LIN {X 0,Y 611.244,Z 977.53,A -85,B 0,C 180,E1 7676.81,E2 7676.81} C_VEL
LIN {X 0,Y 611.181,Z 977.53,A -85,B 0,C 180,E1 7682.54,E2 7682.54} C_VEL
LIN {X 0,Y 611.095,Z 977.53,A -85,B 0,C 180,E1 7688.3,E2 7688.3} C_VEL
LIN {X 0,Y 611.106,Z 977.53,A -85,B 0,C 180,E1 7694.015,E2 7694.015} C_VEL
LIN {X 0,Y 611.087,Z 977.53,A -85,B 0,C 180,E1 7700.225,E2 7700.225} C_VEL
LIN {X 0,Y 611.05,Z 977.53,A -85,B 0,C 180,E1 7705.218,E2 7705.218} C_VEL
LIN {X 0,Y 611.356,Z 977.53,A -85,B 0,C 180,E1 7711.287,E2 7711.287} C_VEL
LIN {X 0,Y 625.159,Z 1016.829,A -85,B 0,C 180,E1 7712.531,E2 7712.531} C_VEL
LIN {X 0,Y 623.748,Z 1056.325,A -85,B 0,C 180,E1 7713.584,E2 7713.584} C_VEL
LIN {X 0,Y 621.786,Z 1092.605,A -85,B 0,C 180,E1 7715.073,E2 7715.073} C_VEL
LIN {X 0,Y 619.511,Z 1127.087,A -85,B 0,C 180,E1 7717.049,E2 7717.049} C_VEL
LIN {X 0,Y 617.19,Z 1158.439,A -85,B 0,C 180,E1 7719.455,E2 7719.455} C_VEL
LIN {X 0,Y 615.112,Z 1187.568,A -85,B 0,C 180,E1 7722.428,E2 7722.428} C_VEL
LIN {X 0,Y 613.624,Z 1211.374,A -85,B 0,C 180,E1 7725.695,E2 7725.695} C_VEL
LIN {X 0,Y 612.633,Z 1230.256,A -85,B 0,C 180,E1 7729.301,E2 7729.301} C_VEL
LIN {X 0,Y 612.205,Z 1242.892,A -85,B 0,C 180,E1 7732.882,E2 7732.882} C_VEL
LIN {X 0,Y 612.031,Z 1249.086,A -85,B 0,C 180,E1 7735.731,E2 7735.731} C_VEL
LIN {X 0,Y 612.003,Z 1252.15,A -85,B 0,C 180,E1 7738.571,E2 7738.571} C_VEL
LIN {X 0,Y 612.141,Z 1252.095,A -85,B 0,C 180,E1 7741.408,E2 7741.408} C_VEL
LIN {X 0,Y 612.201,Z 1247.774,A -85,B 0,C 180,E1 7744.959,E2 7744.959} C_VEL
LIN {X 0,Y 612.397,Z 1238.388,A -85,B 0,C 180,E1 7748.526,E2 7748.526} C_VEL
LIN {X 0,Y 612.998,Z 1222.369,A -85,B 0,C 180,E1 7752.291,E2 7752.291} C_VEL
LIN {X 0,Y 614.182,Z 1202.539,A -85,B 0,C 180,E1 7755.551,E2 7755.551} C_VEL
LIN {X 0,Y 615.818,Z 1177.097,A -85,B 0,C 180,E1 7758.642,E2 7758.642} C_VEL
LIN {X 0,Y 617.854,Z 1148.189,A -85,B 0,C 180,E1 7761.28,E2 7761.28} C_VEL
LIN {X 0,Y 620.03,Z 1114.997,A -85,B 0,C 180,E1 7763.553,E2 7763.553} C_VEL
LIN {X 0,Y 622.154,Z 1077.81,A -85,B 0,C 180,E1 7765.402,E2 7765.402} C_VEL
LIN {X 0,Y 623.879,Z 1037.397,A -85,B 0,C 180,E1 7766.756,E2 7766.756} C_VEL
LIN {X 0,Y 623.911,Z 1015.287,A -85,B 0,C 180,E1 7767.268,E2 7767.268} C_VEL
LIN {X 0,Y 611.262,Z 977.53,A -85,B 0,C 180,E1 7768.438,E2 7768.438} C_VEL
LIN {X 0,Y 611.055,Z 977.53,A -85,B 0,C 180,E1 7774.047,E2 7774.047} C_VEL
LIN {X 0,Y 607.146,Z 977.53,A -85,B 0,C 180,E1 7775.649,E2 7775.649} C_VEL
LIN {X 0,Y 603.114,Z 977.53,A -85,B 0,C 180,E1 7777.271,E2 7777.271} C_VEL
LIN {X 0,Y 602.965,Z 977.53,A -85,B 0,C 180,E1 7783.226,E2 7783.226} C_VEL
LIN {X 0,Y 603.021,Z 977.53,A -85,B 0,C 180,E1 7789.216,E2 7789.216} C_VEL
LIN {X 0,Y 603.25,Z 977.53,A -85,B 0,C 180,E1 7794.718,E2 7794.718} C_VEL
LIN {X 0,Y 603.286,Z 978.056,A -85,B 0,C 180,E1 7798.731,E2 7798.731} C_VEL
LIN {X 0,Y 614.334,Z 1020.655,A -85,B 0,C 180,E1 7801.57,E2 7801.57} C_VEL
LIN {X 0,Y 617.712,Z 1027.362,A -85,B 0,C 180,E1 7801.794,E2 7801.794} C_VEL
LIN {X 0,Y 616.69,Z 1077.628,A -85,B 0,C 180,E1 7802.575,E2 7802.575} C_VEL
LIN {X 0,Y 614.875,Z 1118.446,A -85,B 0,C 180,E1 7803.772,E2 7803.772} C_VEL
LIN {X 0,Y 612.716,Z 1155.496,A -85,B 0,C 180,E1 7805.411,E2 7805.411} C_VEL
LIN {X 0,Y 610.412,Z 1190.848,A -85,B 0,C 180,E1 7807.57,E2 7807.57} C_VEL
LIN {X 0,Y 608.203,Z 1224.713,A -85,B 0,C 180,E1 7810.353,E2 7810.353} C_VEL
LIN {X 0,Y 606.411,Z 1253.135,A -85,B 0,C 180,E1 7813.494,E2 7813.494} C_VEL
LIN {X 0,Y 605.216,Z 1275.601,A -85,B 0,C 180,E1 7816.8,E2 7816.8} C_VEL
LIN {X 0,Y 604.571,Z 1292.527,A -85,B 0,C 180,E1 7820.267,E2 7820.267} C_VEL
LIN {X 0,Y 604.307,Z 1303.392,A -85,B 0,C 180,E1 7823.528,E2 7823.528} C_VEL
LIN {X 0,Y 604.191,Z 1310.148,A -85,B 0,C 180,E1 7827.132,E2 7827.132} C_VEL
LIN {X 0,Y 604.162,Z 1311.816,A -85,B 0,C 180,E1 7830.007,E2 7830.007} C_VEL
LIN {X 0,Y 604.16,Z 1309.117,A -85,B 0,C 180,E1 7833.602,E2 7833.602} C_VEL
LIN {X 0,Y 604.353,Z 1301.231,A -85,B 0,C 180,E1 7837.208,E2 7837.208} C_VEL
LIN {X 0,Y 604.717,Z 1289.245,A -85,B 0,C 180,E1 7840.474,E2 7840.474} C_VEL
LIN {X 0,Y 605.539,Z 1270.525,A -85,B 0,C 180,E1 7843.944,E2 7843.944} C_VEL
LIN {X 0,Y 606.897,Z 1245.039,A -85,B 0,C 180,E1 7847.441,E2 7847.441} C_VEL
LIN {X 0,Y 608.897,Z 1215.102,A -85,B 0,C 180,E1 7850.51,E2 7850.51} C_VEL
LIN {X 0,Y 611.057,Z 1182.798,A -85,B 0,C 180,E1 7852.996,E2 7852.996} C_VEL
LIN {X 0,Y 613.398,Z 1147.018,A -85,B 0,C 180,E1 7855.041,E2 7855.041} C_VEL
LIN {X 0,Y 615.534,Z 1108.168,A -85,B 0,C 180,E1 7856.605,E2 7856.605} C_VEL
LIN {X 0,Y 617.049,Z 1069.386,A -85,B 0,C 180,E1 7857.595,E2 7857.595} C_VEL
LIN {X 0,Y 617.131,Z 1025.386,A -85,B 0,C 180,E1 7858.25,E2 7858.25} C_VEL
LIN {X 0,Y 609.111,Z 1006.368,A -85,B 0,C 180,E1 7858.929,E2 7858.929} C_VEL
LIN {X 0,Y 603.325,Z 977.53,A -85,B 0,C 180,E1 7860.768,E2 7860.768} C_VEL
LIN {X 0,Y 603.185,Z 977.53,A -85,B 0,C 180,E1 7866.525,E2 7866.525} C_VEL
LIN {X 0,Y 603.127,Z 977.53,A -85,B 0,C 180,E1 7871.111,E2 7871.111} C_VEL
LIN {X 0,Y 603.121,Z 977.53,A -85,B 0,C 180,E1 7876.778,E2 7876.778} C_VEL
LIN {X 0,Y 603.127,Z 977.53,A -85,B 0,C 180,E1 7881.164,E2 7881.164} C_VEL
LIN {X 0,Y 603.141,Z 977.53,A -85,B 0,C 180,E1 7886.464,E2 7886.464} C_VEL
LIN {X 0,Y 603.328,Z 977.53,A -85,B 0,C 180,E1 7891.539,E2 7891.539} C_VEL
LIN {X 0,Y 603.432,Z 977.53,A -85,B 0,C 180,E1 7896.325,E2 7896.325} C_VEL
LIN {X 0,Y 603.526,Z 977.53,A -85,B 0,C 180,E1 7900.963,E2 7900.963} C_VEL
LIN {X 0,Y 603.545,Z 977.53,A -85,B 0,C 180,E1 7905.472,E2 7905.472} C_VEL
LIN {X 0,Y 603.751,Z 977.53,A -85,B 0,C 180,E1 7911.351,E2 7911.351} C_VEL
LIN {X 0,Y 603.871,Z 977.53,A -85,B 0,C 180,E1 7913.437,E2 7913.437} C_VEL
LIN {X 0,Y 611.206,Z 1003.096,A -85,B 0,C 180,E1 7914.239,E2 7914.239} C_VEL
LIN {X 0,Y 610.052,Z 1060.493,A -85,B 0,C 180,E1 7915.336,E2 7915.336} C_VEL
LIN {X 0,Y 609.176,Z 1088.907,A -85,B 0,C 180,E1 7916.445,E2 7916.445} C_VEL
LIN {X 0,Y 608.114,Z 1114.127,A -85,B 0,C 180,E1 7918.047,E2 7918.047} C_VEL
LIN {X 0,Y 606.979,Z 1135.109,A -85,B 0,C 180,E1 7920.01,E2 7920.01} C_VEL
LIN {X 0,Y 606.057,Z 1152.124,A -85,B 0,C 180,E1 7922.338,E2 7922.338} C_VEL
LIN {X 0,Y 605.342,Z 1164.6,A -85,B 0,C 180,E1 7925.036,E2 7925.036} C_VEL
LIN {X 0,Y 605.013,Z 1170.296,A -85,B 0,C 180,E1 7927.203,E2 7927.203} C_VEL
LIN {X 0,Y 604.838,Z 1172.559,A -85,B 0,C 180,E1 7930.109,E2 7930.109} C_VEL
LIN {X 0,Y 604.97,Z 1168.797,A -85,B 0,C 180,E1 7933.037,E2 7933.037} C_VEL
LIN {X 0,Y 605.309,Z 1159.648,A -85,B 0,C 180,E1 7935.744,E2 7935.744} C_VEL
LIN {X 0,Y 605.903,Z 1145.613,A -85,B 0,C 180,E1 7938.203,E2 7938.203} C_VEL
LIN {X 0,Y 606.787,Z 1126.099,A -85,B 0,C 180,E1 7940.472,E2 7940.472} C_VEL
LIN {X 0,Y 607.731,Z 1102.106,A -85,B 0,C 180,E1 7942.367,E2 7942.367} C_VEL
LIN {X 0,Y 608.82,Z 1074.436,A -85,B 0,C 180,E1 7943.782,E2 7943.782} C_VEL
LIN {X 0,Y 609.304,Z 1045.453,A -85,B 0,C 180,E1 7944.644,E2 7944.644} C_VEL
LIN {X 0,Y 609.265,Z 999.333,A -85,B 0,C 180,E1 7945.356,E2 7945.356} C_VEL
LIN {X 0,Y 603.556,Z 977.53,A -85,B 0,C 180,E1 7945.917,E2 7945.917} C_VEL
LIN {X 0,Y 603.26,Z 977.53,A -85,B 0,C 180,E1 7951.843,E2 7951.843} C_VEL
LIN {X 0,Y 603.173,Z 977.53,A -85,B 0,C 180,E1 7957.087,E2 7957.087} C_VEL
LIN {X 0,Y 603.145,Z 977.53,A -85,B 0,C 180,E1 7962.72,E2 7962.72} C_VEL
LIN {X 0,Y 603.092,Z 977.53,A -85,B 0,C 180,E1 7967.274,E2 7967.274} C_VEL
LIN {X 0,Y 603.118,Z 977.53,A -85,B 0,C 180,E1 7972.909,E2 7972.909} C_VEL
LIN {X 0,Y 603.263,Z 977.53,A -85,B 0,C 180,E1 7978.659,E2 7978.659} C_VEL
LIN {X 0,Y 603.392,Z 977.53,A -85,B 0,C 180,E1 7983.119,E2 7983.119} C_VEL
LIN {X 0,Y 603.49,Z 977.53,A -85,B 0,C 180,E1 7988.291,E2 7988.291} C_VEL
LIN {X 0,Y 603.561,Z 977.53,A -85,B 0,C 180,E1 7993.962,E2 7993.962} C_VEL
LIN {X 0,Y 603.681,Z 977.53,A -85,B 0,C 180,E1 7999.874,E2 7999.874} C_VEL
LIN {X 0,Y 603.86,Z 977.53,A -85,B 0,C 180,E1 8004.233,E2 8004.233} C_VEL
LIN {X 0,Y 603.917,Z 977.53,A -85,B 0,C 180,E1 8008.556,E2 8008.556} C_VEL
LIN {X 0,Y 603.938,Z 977.53,A -85,B 0,C 180,E1 8012.87,E2 8012.87} C_VEL
LIN {X 0,Y 603.718,Z 977.53,A -85,B 0,C 180,E1 8017.203,E2 8017.203} C_VEL
LIN {X 0,Y 603.623,Z 977.53,A -85,B 0,C 180,E1 8023.05,E2 8023.05} C_VEL
LIN {X 0,Y 603.572,Z 977.53,A -85,B 0,C 180,E1 8027.526,E2 8027.526} C_VEL
LIN {X 0,Y 603.428,Z 977.53,A -85,B 0,C 180,E1 8032.12,E2 8032.12} C_VEL
LIN {X 0,Y 603.363,Z 977.53,A -85,B 0,C 180,E1 8036.867,E2 8036.867} C_VEL
LIN {X 0,Y 603.267,Z 977.53,A -85,B 0,C 180,E1 8041.827,E2 8041.827} C_VEL
LIN {X 0,Y 603.174,Z 977.53,A -85,B 0,C 180,E1 8047.071,E2 8047.071} C_VEL
LIN {X 0,Y 603.135,Z 977.53,A -85,B 0,C 180,E1 8052.704,E2 8052.704} C_VEL
LIN {X 0,Y 603.086,Z 977.53,A -85,B 0,C 180,E1 8057.275,E2 8057.275} C_VEL
LIN {X 0,Y 603.127,Z 977.53,A -85,B 0,C 180,E1 8062.91,E2 8062.91} C_VEL
LIN {X 0,Y 603.264,Z 977.53,A -85,B 0,C 180,E1 8068.637,E2 8068.637} C_VEL
LIN {X 0,Y 603.415,Z 977.689,A -85,B 0,C 180,E1 8070.929,E2 8070.929} C_VEL
LIN {X 0,Y 617.942,Z 1019.384,A -85,B 0,C 180,E1 8072.271,E2 8072.271} C_VEL
LIN {X 0,Y 616.402,Z 1059.794,A -85,B 0,C 180,E1 8073.401,E2 8073.401} C_VEL
LIN {X 0,Y 614.144,Z 1097.737,A -85,B 0,C 180,E1 8075.035,E2 8075.035} C_VEL
LIN {X 0,Y 611.585,Z 1133.527,A -85,B 0,C 180,E1 8077.216,E2 8077.216} C_VEL
LIN {X 0,Y 609.219,Z 1164.975,A -85,B 0,C 180,E1 8079.804,E2 8079.804} C_VEL
LIN {X 0,Y 607.126,Z 1192.049,A -85,B 0,C 180,E1 8082.751,E2 8082.751} C_VEL
LIN {X 0,Y 605.697,Z 1213.671,A -85,B 0,C 180,E1 8085.873,E2 8085.873} C_VEL
LIN {X 0,Y 604.809,Z 1230.485,A -85,B 0,C 180,E1 8089.161,E2 8089.161} C_VEL
LIN {X 0,Y 604.345,Z 1243.19,A -85,B 0,C 180,E1 8092.789,E2 8092.789} C_VEL
LIN {X 0,Y 604.146,Z 1249.426,A -85,B 0,C 180,E1 8095.675,E2 8095.675} C_VEL
LIN {X 0,Y 604.112,Z 1252.516,A -85,B 0,C 180,E1 8098.553,E2 8098.553} C_VEL
LIN {X 0,Y 604.266,Z 1252.471,A -85,B 0,C 180,E1 8101.426,E2 8101.426} C_VEL
LIN {X 0,Y 604.313,Z 1248.139,A -85,B 0,C 180,E1 8105.024,E2 8105.024} C_VEL
LIN {X 0,Y 604.545,Z 1238.716,A -85,B 0,C 180,E1 8108.638,E2 8108.638} C_VEL
LIN {X 0,Y 605.162,Z 1223.209,A -85,B 0,C 180,E1 8112.336,E2 8112.336} C_VEL
LIN {X 0,Y 606.453,Z 1202.656,A -85,B 0,C 180,E1 8115.754,E2 8115.754} C_VEL
LIN {X 0,Y 608.146,Z 1177.906,A -85,B 0,C 180,E1 8118.792,E2 8118.792} C_VEL
LIN {X 0,Y 610.342,Z 1148.346,A -85,B 0,C 180,E1 8121.519,E2 8121.519} C_VEL
LIN {X 0,Y 612.598,Z 1114.641,A -85,B 0,C 180,E1 8123.844,E2 8123.844} C_VEL
LIN {X 0,Y 614.838,Z 1077.728,A -85,B 0,C 180,E1 8125.689,E2 8125.689} C_VEL
LIN {X 0,Y 616.627,Z 1037.109,A -85,B 0,C 180,E1 8127.056,E2 8127.056} C_VEL
LIN {X 0,Y 616.657,Z 1017.258,A -85,B 0,C 180,E1 8127.528,E2 8127.528} C_VEL
LIN {X 0,Y 603.35,Z 977.53,A -85,B 0,C 180,E1 8128.823,E2 8128.823} C_VEL
LIN {X 0,Y 603.163,Z 977.53,A -85,B 0,C 180,E1 8134.041,E2 8134.041} C_VEL
LIN {X 0,Y 603.114,Z 977.53,A -85,B 0,C 180,E1 8137.271,E2 8137.271} C_VEL
LIN {X 0,Y 599.073,Z 977.53,A -85,B 0,C 180,E1 8138.893,E2 8138.893} C_VEL
LIN {X 0,Y 595.066,Z 977.53,A -85,B 0,C 180,E1 8140.535,E2 8140.535} C_VEL
LIN {X 0,Y 595.061,Z 977.53,A -85,B 0,C 180,E1 8145.457,E2 8145.457} C_VEL
LIN {X 0,Y 595.116,Z 977.53,A -85,B 0,C 180,E1 8150.474,E2 8150.474} C_VEL
LIN {X 0,Y 595.331,Z 977.53,A -85,B 0,C 180,E1 8155.956,E2 8155.956} C_VEL
LIN {X 0,Y 595.329,Z 977.778,A -85,B 0,C 180,E1 8158.372,E2 8158.372} C_VEL
LIN {X 0,Y 606.071,Z 1020.674,A -85,B 0,C 180,E1 8161.23,E2 8161.23} C_VEL
LIN {X 0,Y 610.515,Z 1031.2,A -85,B 0,C 180,E1 8161.553,E2 8161.553} C_VEL
LIN {X 0,Y 609.35,Z 1077.574,A -85,B 0,C 180,E1 8162.301,E2 8162.301} C_VEL
LIN {X 0,Y 607.51,Z 1117.465,A -85,B 0,C 180,E1 8163.485,E2 8163.485} C_VEL
LIN {X 0,Y 605.122,Z 1155.894,A -85,B 0,C 180,E1 8165.209,E2 8165.209} C_VEL
LIN {X 0,Y 602.651,Z 1191.864,A -85,B 0,C 180,E1 8167.461,E2 8167.461} C_VEL
LIN {X 0,Y 600.576,Z 1223.393,A -85,B 0,C 180,E1 8170.093,E2 8170.093} C_VEL
LIN {X 0,Y 598.666,Z 1251.991,A -85,B 0,C 180,E1 8173.274,E2 8173.274} C_VEL
LIN {X 0,Y 597.407,Z 1274.588,A -85,B 0,C 180,E1 8176.625,E2 8176.625} C_VEL
LIN {X 0,Y 596.722,Z 1291.588,A -85,B 0,C 180,E1 8180.137,E2 8180.137} C_VEL
LIN {X 0,Y 596.439,Z 1302.503,A -85,B 0,C 180,E1 8183.442,E2 8183.442} C_VEL
LIN {X 0,Y 596.341,Z 1309.289,A -85,B 0,C 180,E1 8187.094,E2 8187.094} C_VEL
LIN {X 0,Y 596.316,Z 1310.95,A -85,B 0,C 180,E1 8190.007,E2 8190.007} C_VEL
LIN {X 0,Y 596.322,Z 1308.212,A -85,B 0,C 180,E1 8193.649,E2 8193.649} C_VEL
LIN {X 0,Y 596.524,Z 1300.246,A -85,B 0,C 180,E1 8197.304,E2 8197.304} C_VEL
LIN {X 0,Y 596.853,Z 1288.156,A -85,B 0,C 180,E1 8200.613,E2 8200.613} C_VEL
LIN {X 0,Y 597.753,Z 1267.354,A -85,B 0,C 180,E1 8204.504,E2 8204.504} C_VEL
LIN {X 0,Y 599.211,Z 1243.275,A -85,B 0,C 180,E1 8207.81,E2 8207.81} C_VEL
LIN {X 0,Y 601.274,Z 1213.743,A -85,B 0,C 180,E1 8210.833,E2 8210.833} C_VEL
LIN {X 0,Y 603.708,Z 1180.457,A -85,B 0,C 180,E1 8213.391,E2 8213.391} C_VEL
LIN {X 0,Y 606.121,Z 1145.205,A -85,B 0,C 180,E1 8215.399,E2 8215.399} C_VEL
LIN {X 0,Y 608.335,Z 1106.849,A -85,B 0,C 180,E1 8216.939,E2 8216.939} C_VEL
LIN {X 0,Y 609.968,Z 1067.091,A -85,B 0,C 180,E1 8217.943,E2 8217.943} C_VEL
LIN {X 0,Y 610.095,Z 1027.985,A -85,B 0,C 180,E1 8218.527,E2 8218.527} C_VEL
LIN {X 0,Y 600.85,Z 1004.137,A -85,B 0,C 180,E1 8219.353,E2 8219.353} C_VEL
LIN {X 0,Y 595.426,Z 977.53,A -85,B 0,C 180,E1 8221.124,E2 8221.124} C_VEL
LIN {X 0,Y 595.257,Z 977.53,A -85,B 0,C 180,E1 8225.845,E2 8225.845} C_VEL
LIN {X 0,Y 595.206,Z 977.53,A -85,B 0,C 180,E1 8231.454,E2 8231.454} C_VEL
LIN {X 0,Y 595.22,Z 977.53,A -85,B 0,C 180,E1 8236.6,E2 8236.6} C_VEL
LIN {X 0,Y 595.155,Z 977.53,A -85,B 0,C 180,E1 8242.354,E2 8242.354} C_VEL
LIN {X 0,Y 595.256,Z 977.53,A -85,B 0,C 180,E1 8247.702,E2 8247.702} C_VEL
LIN {X 0,Y 595.492,Z 977.53,A -85,B 0,C 180,E1 8252.963,E2 8252.963} C_VEL
LIN {X 0,Y 595.526,Z 977.53,A -85,B 0,C 180,E1 8257.577,E2 8257.577} C_VEL
LIN {X 0,Y 595.598,Z 977.53,A -85,B 0,C 180,E1 8262.237,E2 8262.237} C_VEL
LIN {X 0,Y 595.618,Z 977.53,A -85,B 0,C 180,E1 8266.776,E2 8266.776} C_VEL
LIN {X 0,Y 595.916,Z 977.53,A -85,B 0,C 180,E1 8272.707,E2 8272.707} C_VEL
LIN {X 0,Y 595.959,Z 977.53,A -85,B 0,C 180,E1 8273.075,E2 8273.075} C_VEL
LIN {X 0,Y 603.888,Z 1005.096,A -85,B 0,C 180,E1 8273.984,E2 8273.984} C_VEL
LIN {X 0,Y 602.566,Z 1062.313,A -85,B 0,C 180,E1 8275.126,E2 8275.126} C_VEL
LIN {X 0,Y 601.696,Z 1089.668,A -85,B 0,C 180,E1 8276.22,E2 8276.22} C_VEL
LIN {X 0,Y 600.541,Z 1114.948,A -85,B 0,C 180,E1 8277.842,E2 8277.842} C_VEL
LIN {X 0,Y 599.239,Z 1137.543,A -85,B 0,C 180,E1 8280.01,E2 8280.01} C_VEL
LIN {X 0,Y 598.228,Z 1154.978,A -85,B 0,C 180,E1 8282.551,E2 8282.551} C_VEL
LIN {X 0,Y 597.515,Z 1166.087,A -85,B 0,C 180,E1 8285.102,E2 8285.102} C_VEL
LIN {X 0,Y 597.169,Z 1171.546,A -85,B 0,C 180,E1 8287.298,E2 8287.298} C_VEL
LIN {X 0,Y 596.991,Z 1173.453,A -85,B 0,C 180,E1 8290.244,E2 8290.244} C_VEL
LIN {X 0,Y 597.158,Z 1169.391,A -85,B 0,C 180,E1 8293.21,E2 8293.21} C_VEL
LIN {X 0,Y 597.519,Z 1159.721,A -85,B 0,C 180,E1 8295.984,E2 8295.984} C_VEL
LIN {X 0,Y 598.219,Z 1144.574,A -85,B 0,C 180,E1 8298.565,E2 8298.565} C_VEL
LIN {X 0,Y 599.174,Z 1124.452,A -85,B 0,C 180,E1 8300.841,E2 8300.841} C_VEL
LIN {X 0,Y 600.182,Z 1100.359,A -85,B 0,C 180,E1 8302.682,E2 8302.682} C_VEL
LIN {X 0,Y 601.226,Z 1072.101,A -85,B 0,C 180,E1 8304.086,E2 8304.086} C_VEL
LIN {X 0,Y 601.73,Z 1041.841,A -85,B 0,C 180,E1 8304.921,E2 8304.921} C_VEL
LIN {X 0,Y 601.803,Z 1001.087,A -85,B 0,C 180,E1 8305.551,E2 8305.551} C_VEL
LIN {X 0,Y 595.614,Z 977.53,A -85,B 0,C 180,E1 8306.157,E2 8306.157} C_VEL
LIN {X 0,Y 595.293,Z 977.53,A -85,B 0,C 180,E1 8312.32,E2 8312.32} C_VEL
LIN {X 0,Y 595.207,Z 977.53,A -85,B 0,C 180,E1 8317.879,E2 8317.879} C_VEL
LIN {X 0,Y 595.266,Z 977.53,A -85,B 0,C 180,E1 8323.424,E2 8323.424} C_VEL
LIN {X 0,Y 595.15,Z 977.53,A -85,B 0,C 180,E1 8328.541,E2 8328.541} C_VEL
LIN {X 0,Y 595.211,Z 977.53,A -85,B 0,C 180,E1 8334.56,E2 8334.56} C_VEL
LIN {X 0,Y 595.367,Z 977.53,A -85,B 0,C 180,E1 8339.93,E2 8339.93} C_VEL
LIN {X 0,Y 595.493,Z 977.53,A -85,B 0,C 180,E1 8344.362,E2 8344.362} C_VEL
LIN {X 0,Y 595.552,Z 977.53,A -85,B 0,C 180,E1 8349.126,E2 8349.126} C_VEL
LIN {X 0,Y 595.639,Z 977.53,A -85,B 0,C 180,E1 8353.743,E2 8353.743} C_VEL
LIN {X 0,Y 595.789,Z 977.53,A -85,B 0,C 180,E1 8359.738,E2 8359.738} C_VEL
LIN {X 0,Y 595.949,Z 977.53,A -85,B 0,C 180,E1 8364.156,E2 8364.156} C_VEL
LIN {X 0,Y 596.016,Z 977.53,A -85,B 0,C 180,E1 8368.536,E2 8368.536} C_VEL
LIN {X 0,Y 596.034,Z 977.53,A -85,B 0,C 180,E1 8372.908,E2 8372.908} C_VEL
LIN {X 0,Y 595.818,Z 977.53,A -85,B 0,C 180,E1 8377.299,E2 8377.299} C_VEL
LIN {X 0,Y 595.752,Z 977.53,A -85,B 0,C 180,E1 8381.733,E2 8381.733} C_VEL
LIN {X 0,Y 595.657,Z 977.53,A -85,B 0,C 180,E1 8386.243,E2 8386.243} C_VEL
LIN {X 0,Y 595.544,Z 977.53,A -85,B 0,C 180,E1 8390.86,E2 8390.86} C_VEL
LIN {X 0,Y 595.44,Z 977.53,A -85,B 0,C 180,E1 8395.626,E2 8395.626} C_VEL
LIN {X 0,Y 595.346,Z 977.53,A -85,B 0,C 180,E1 8400.592,E2 8400.592} C_VEL
LIN {X 0,Y 595.271,Z 977.53,A -85,B 0,C 180,E1 8405.827,E2 8405.827} C_VEL
LIN {X 0,Y 595.217,Z 977.53,A -85,B 0,C 180,E1 8411.435,E2 8411.435} C_VEL
LIN {X 0,Y 595.205,Z 977.53,A -85,B 0,C 180,E1 8416.57,E2 8416.57} C_VEL
LIN {X 0,Y 595.161,Z 977.53,A -85,B 0,C 180,E1 8422.328,E2 8422.328} C_VEL
LIN {X 0,Y 595.258,Z 977.53,A -85,B 0,C 180,E1 8427.677,E2 8427.677} C_VEL
LIN {X 0,Y 595.484,Z 978.235,A -85,B 0,C 180,E1 8430.561,E2 8430.561} C_VEL
LIN {X 0,Y 610.794,Z 1020.179,A -85,B 0,C 180,E1 8431.972,E2 8431.972} C_VEL
LIN {X 0,Y 609.136,Z 1060.705,A -85,B 0,C 180,E1 8433.125,E2 8433.125} C_VEL
LIN {X 0,Y 606.683,Z 1100.08,A -85,B 0,C 180,E1 8434.867,E2 8434.867} C_VEL
LIN {X 0,Y 603.985,Z 1135.793,A -85,B 0,C 180,E1 8437.108,E2 8437.108} C_VEL
LIN {X 0,Y 601.486,Z 1166.793,A -85,B 0,C 180,E1 8439.725,E2 8439.725} C_VEL
LIN {X 0,Y 599.341,Z 1193.534,A -85,B 0,C 180,E1 8442.71,E2 8442.71} C_VEL
LIN {X 0,Y 597.772,Z 1215.966,A -85,B 0,C 180,E1 8446.057,E2 8446.057} C_VEL
LIN {X 0,Y 596.898,Z 1232.234,A -85,B 0,C 180,E1 8449.385,E2 8449.385} C_VEL
LIN {X 0,Y 596.484,Z 1243.49,A -85,B 0,C 180,E1 8452.693,E2 8452.693} C_VEL
LIN {X 0,Y 596.26,Z 1249.76,A -85,B 0,C 180,E1 8455.618,E2 8455.618} C_VEL
LIN {X 0,Y 596.22,Z 1252.88,A -85,B 0,C 180,E1 8458.533,E2 8458.533} C_VEL
LIN {X 0,Y 596.374,Z 1252.848,A -85,B 0,C 180,E1 8461.445,E2 8461.445} C_VEL
LIN {X 0,Y 596.441,Z 1248.502,A -85,B 0,C 180,E1 8465.09,E2 8465.09} C_VEL
LIN {X 0,Y 596.68,Z 1239.038,A -85,B 0,C 180,E1 8468.753,E2 8468.753} C_VEL
LIN {X 0,Y 597.347,Z 1223.864,A -85,B 0,C 180,E1 8472.419,E2 8472.419} C_VEL
LIN {X 0,Y 598.7,Z 1203.041,A -85,B 0,C 180,E1 8475.923,E2 8475.923} C_VEL
LIN {X 0,Y 600.471,Z 1178.109,A -85,B 0,C 180,E1 8479.014,E2 8479.014} C_VEL
LIN {X 0,Y 602.798,Z 1148.747,A -85,B 0,C 180,E1 8481.747,E2 8481.747} C_VEL
LIN {X 0,Y 605.16,Z 1115.407,A -85,B 0,C 180,E1 8484.077,E2 8484.077} C_VEL
LIN {X 0,Y 607.558,Z 1077.623,A -85,B 0,C 180,E1 8485.989,E2 8485.989} C_VEL
LIN {X 0,Y 609.443,Z 1036.846,A -85,B 0,C 180,E1 8487.368,E2 8487.368} C_VEL
LIN {X 0,Y 609.292,Z 1018.723,A -85,B 0,C 180,E1 8487.817,E2 8487.817} C_VEL
LIN {X 0,Y 595.404,Z 977.53,A -85,B 0,C 180,E1 8489.232,E2 8489.232} C_VEL
LIN {X 0,Y 595.264,Z 977.53,A -85,B 0,C 180,E1 8494.04,E2 8494.04} C_VEL
LIN {X 0,Y 595.122,Z 977.53,A -85,B 0,C 180,E1 8499.515,E2 8499.515} C_VEL
LIN {X 0,Y 595.066,Z 977.53,A -85,B 0,C 180,E1 8500.535,E2 8500.535} C_VEL
LIN {X 0,Y 591.085,Z 977.53,A -85,B 0,C 180,E1 8502.178,E2 8502.178} C_VEL
LIN {X 0,Y 587.14,Z 977.53,A -85,B 0,C 180,E1 8503.843,E2 8503.843} C_VEL
LIN {X 0,Y 587.203,Z 977.53,A -85,B 0,C 180,E1 8509.835,E2 8509.835} C_VEL
LIN {X 0,Y 587.423,Z 977.53,A -85,B 0,C 180,E1 8515.605,E2 8515.605} C_VEL
LIN {X 0,Y 587.468,Z 978.239,A -85,B 0,C 180,E1 8518.056,E2 8518.056} C_VEL
LIN {X 0,Y 597.814,Z 1020.503,A -85,B 0,C 180,E1 8520.88,E2 8520.88} C_VEL
LIN {X 0,Y 603.229,Z 1033.307,A -85,B 0,C 180,E1 8521.284,E2 8521.284} C_VEL
LIN {X 0,Y 601.982,Z 1078.358,A -85,B 0,C 180,E1 8522.04,E2 8522.04} C_VEL
LIN {X 0,Y 600.052,Z 1117.57,A -85,B 0,C 180,E1 8523.234,E2 8523.234} C_VEL
LIN {X 0,Y 597.545,Z 1155.69,A -85,B 0,C 180,E1 8524.973,E2 8524.973} C_VEL
LIN {X 0,Y 595.104,Z 1190.725,A -85,B 0,C 180,E1 8527.189,E2 8527.189} C_VEL
LIN {X 0,Y 592.88,Z 1222.045,A -85,B 0,C 180,E1 8529.824,E2 8529.824} C_VEL
LIN {X 0,Y 591.005,Z 1249.369,A -85,B 0,C 180,E1 8532.859,E2 8532.859} C_VEL
LIN {X 0,Y 589.653,Z 1272.508,A -85,B 0,C 180,E1 8536.256,E2 8536.256} C_VEL
LIN {X 0,Y 588.917,Z 1289.152,A -85,B 0,C 180,E1 8539.631,E2 8539.631} C_VEL
LIN {X 0,Y 588.582,Z 1301.614,A -85,B 0,C 180,E1 8543.354,E2 8543.354} C_VEL
LIN {X 0,Y 588.49,Z 1308.43,A -85,B 0,C 180,E1 8547.055,E2 8547.055} C_VEL
LIN {X 0,Y 588.491,Z 1310.085,A -85,B 0,C 180,E1 8550.007,E2 8550.007} C_VEL
LIN {X 0,Y 588.488,Z 1307.312,A -85,B 0,C 180,E1 8553.698,E2 8553.698} C_VEL
LIN {X 0,Y 588.682,Z 1299.282,A -85,B 0,C 180,E1 8557.401,E2 8557.401} C_VEL
LIN {X 0,Y 589.042,Z 1285.709,A -85,B 0,C 180,E1 8561.131,E2 8561.131} C_VEL
LIN {X 0,Y 589.991,Z 1265.673,A -85,B 0,C 180,E1 8564.889,E2 8564.889} C_VEL
LIN {X 0,Y 591.557,Z 1242.039,A -85,B 0,C 180,E1 8568.118,E2 8568.118} C_VEL
LIN {X 0,Y 593.668,Z 1213.313,A -85,B 0,C 180,E1 8571.082,E2 8571.082} C_VEL
LIN {X 0,Y 596.094,Z 1181.744,A -85,B 0,C 180,E1 8573.553,E2 8573.553} C_VEL
LIN {X 0,Y 598.63,Z 1146.744,A -85,B 0,C 180,E1 8575.597,E2 8575.597} C_VEL
LIN {X 0,Y 600.913,Z 1109.412,A -85,B 0,C 180,E1 8577.15,E2 8577.15} C_VEL
LIN {X 0,Y 602.633,Z 1070.989,A -85,B 0,C 180,E1 8578.182,E2 8578.182} C_VEL
LIN {X 0,Y 602.776,Z 1029.877,A -85,B 0,C 180,E1 8578.836,E2 8578.836} C_VEL
LIN {X 0,Y 593.479,Z 1005.645,A -85,B 0,C 180,E1 8579.615,E2 8579.615} C_VEL
LIN {X 0,Y 587.468,Z 977.53,A -85,B 0,C 180,E1 8581.453,E2 8581.453} C_VEL
LIN {X 0,Y 587.279,Z 977.53,A -85,B 0,C 180,E1 8586.911,E2 8586.911} C_VEL
LIN {X 0,Y 587.303,Z 977.53,A -85,B 0,C 180,E1 8592.139,E2 8592.139} C_VEL
LIN {X 0,Y 587.255,Z 977.53,A -85,B 0,C 180,E1 8597.887,E2 8597.887} C_VEL
LIN {X 0,Y 587.229,Z 977.53,A -85,B 0,C 180,E1 8603.614,E2 8603.614} C_VEL
LIN {X 0,Y 587.358,Z 977.53,A -85,B 0,C 180,E1 8608.955,E2 8608.955} C_VEL
LIN {X 0,Y 587.616,Z 977.53,A -85,B 0,C 180,E1 8614.509,E2 8614.509} C_VEL
LIN {X 0,Y 587.691,Z 977.53,A -85,B 0,C 180,E1 8620.43,E2 8620.43} C_VEL
LIN {X 0,Y 587.735,Z 977.53,A -85,B 0,C 180,E1 8625.072,E2 8625.072} C_VEL
LIN {X 0,Y 587.848,Z 977.53,A -85,B 0,C 180,E1 8629.617,E2 8629.617} C_VEL
LIN {X 0,Y 588.038,Z 977.71,A -85,B 0,C 180,E1 8632.705,E2 8632.705} C_VEL
LIN {X 0,Y 596.573,Z 1006.679,A -85,B 0,C 180,E1 8633.712,E2 8633.712} C_VEL
LIN {X 0,Y 595.147,Z 1063.926,A -85,B 0,C 180,E1 8634.899,E2 8634.899} C_VEL
LIN {X 0,Y 594.17,Z 1092.248,A -85,B 0,C 180,E1 8636.081,E2 8636.081} C_VEL
LIN {X 0,Y 592.844,Z 1118.023,A -85,B 0,C 180,E1 8637.814,E2 8637.814} C_VEL
LIN {X 0,Y 591.596,Z 1138.376,A -85,B 0,C 180,E1 8639.827,E2 8639.827} C_VEL
LIN {X 0,Y 590.583,Z 1154.87,A -85,B 0,C 180,E1 8642.216,E2 8642.216} C_VEL
LIN {X 0,Y 589.779,Z 1166.372,A -85,B 0,C 180,E1 8644.8,E2 8644.8} C_VEL
LIN {X 0,Y 589.341,Z 1172.74,A -85,B 0,C 180,E1 8647.396,E2 8647.396} C_VEL
LIN {X 0,Y 589.162,Z 1174.345,A -85,B 0,C 180,E1 8650.381,E2 8650.381} C_VEL
LIN {X 0,Y 589.326,Z 1169.946,A -85,B 0,C 180,E1 8653.389,E2 8653.389} C_VEL
LIN {X 0,Y 589.719,Z 1160.673,A -85,B 0,C 180,E1 8656.038,E2 8656.038} C_VEL
LIN {X 0,Y 590.442,Z 1145.858,A -85,B 0,C 180,E1 8658.609,E2 8658.609} C_VEL
LIN {X 0,Y 591.432,Z 1126.196,A -85,B 0,C 180,E1 8660.888,E2 8660.888} C_VEL
LIN {X 0,Y 592.477,Z 1102.009,A -85,B 0,C 180,E1 8662.792,E2 8662.792} C_VEL
LIN {X 0,Y 593.575,Z 1075.038,A -85,B 0,C 180,E1 8664.182,E2 8664.182} C_VEL
LIN {X 0,Y 594.148,Z 1045.784,A -85,B 0,C 180,E1 8665.061,E2 8665.061} C_VEL
LIN {X 0,Y 594.138,Z 1001.921,A -85,B 0,C 180,E1 8665.77,E2 8665.77} C_VEL
LIN {X 0,Y 587.694,Z 977.53,A -85,B 0,C 180,E1 8666.408,E2 8666.408} C_VEL
LIN {X 0,Y 587.4,Z 977.53,A -85,B 0,C 180,E1 8672.809,E2 8672.809} C_VEL
LIN {X 0,Y 587.272,Z 977.53,A -85,B 0,C 180,E1 8678.269,E2 8678.269} C_VEL
LIN {X 0,Y 587.343,Z 977.53,A -85,B 0,C 180,E1 8684.16,E2 8684.16} C_VEL
LIN {X 0,Y 587.25,Z 977.53,A -85,B 0,C 180,E1 8689.82,E2 8689.82} C_VEL
LIN {X 0,Y 587.308,Z 977.53,A -85,B 0,C 180,E1 8695.659,E2 8695.659} C_VEL
LIN {X 0,Y 587.439,Z 977.53,A -85,B 0,C 180,E1 8701.293,E2 8701.293} C_VEL
LIN {X 0,Y 587.561,Z 977.53,A -85,B 0,C 180,E1 8705.623,E2 8705.623} C_VEL
LIN {X 0,Y 587.666,Z 977.53,A -85,B 0,C 180,E1 8710.408,E2 8710.408} C_VEL
LIN {X 0,Y 587.762,Z 977.53,A -85,B 0,C 180,E1 8715.053,E2 8715.053} C_VEL
LIN {X 0,Y 587.871,Z 977.53,A -85,B 0,C 180,E1 8719.598,E2 8719.598} C_VEL
LIN {X 0,Y 588.044,Z 977.53,A -85,B 0,C 180,E1 8724.077,E2 8724.077} C_VEL
LIN {X 0,Y 588.133,Z 977.53,A -85,B 0,C 180,E1 8728.517,E2 8728.517} C_VEL
LIN {X 0,Y 588.129,Z 977.53,A -85,B 0,C 180,E1 8732.947,E2 8732.947} C_VEL
LIN {X 0,Y 587.907,Z 977.53,A -85,B 0,C 180,E1 8737.397,E2 8737.397} C_VEL
LIN {X 0,Y 587.843,Z 977.53,A -85,B 0,C 180,E1 8741.894,E2 8741.894} C_VEL
LIN {X 0,Y 587.707,Z 977.53,A -85,B 0,C 180,E1 8747.441,E2 8747.441} C_VEL
LIN {X 0,Y 587.558,Z 977.53,A -85,B 0,C 180,E1 8752.75,E2 8752.75} C_VEL
LIN {X 0,Y 587.46,Z 977.53,A -85,B 0,C 180,E1 8757.656,E2 8757.656} C_VEL
LIN {X 0,Y 587.39,Z 977.53,A -85,B 0,C 180,E1 8762.793,E2 8762.793} C_VEL
LIN {X 0,Y 587.27,Z 977.53,A -85,B 0,C 180,E1 8768.252,E2 8768.252} C_VEL
LIN {X 0,Y 587.322,Z 977.53,A -85,B 0,C 180,E1 8774.144,E2 8774.144} C_VEL
LIN {X 0,Y 587.266,Z 977.53,A -85,B 0,C 180,E1 8779.823,E2 8779.823} C_VEL
LIN {X 0,Y 587.32,Z 977.53,A -85,B 0,C 180,E1 8785.636,E2 8785.636} C_VEL
LIN {X 0,Y 587.506,Z 977.53,A -85,B 0,C 180,E1 8790.152,E2 8790.152} C_VEL
LIN {X 0,Y 603.621,Z 1022.516,A -85,B 0,C 180,E1 8791.701,E2 8791.701} C_VEL
LIN {X 0,Y 601.756,Z 1063.712,A -85,B 0,C 180,E1 8792.923,E2 8792.923} C_VEL
LIN {X 0,Y 599.26,Z 1101.232,A -85,B 0,C 180,E1 8794.632,E2 8794.632} C_VEL
LIN {X 0,Y 596.456,Z 1136.791,A -85,B 0,C 180,E1 8796.901,E2 8796.901} C_VEL
LIN {X 0,Y 593.963,Z 1166.69,A -85,B 0,C 180,E1 8799.457,E2 8799.457} C_VEL
LIN {X 0,Y 591.663,Z 1193.567,A -85,B 0,C 180,E1 8802.478,E2 8802.478} C_VEL
LIN {X 0,Y 590.012,Z 1216.103,A -85,B 0,C 180,E1 8805.869,E2 8805.869} C_VEL
LIN {X 0,Y 589.079,Z 1232.46,A -85,B 0,C 180,E1 8809.243,E2 8809.243} C_VEL
LIN {X 0,Y 588.624,Z 1243.785,A -85,B 0,C 180,E1 8812.595,E2 8812.595} C_VEL
LIN {X 0,Y 588.375,Z 1250.101,A -85,B 0,C 180,E1 8815.559,E2 8815.559} C_VEL
LIN {X 0,Y 588.359,Z 1253.245,A -85,B 0,C 180,E1 8818.514,E2 8818.514} C_VEL
LIN {X 0,Y 588.495,Z 1253.225,A -85,B 0,C 180,E1 8821.465,E2 8821.465} C_VEL
LIN {X 0,Y 588.557,Z 1248.865,A -85,B 0,C 180,E1 8825.159,E2 8825.159} C_VEL
LIN {X 0,Y 588.836,Z 1239.357,A -85,B 0,C 180,E1 8828.87,E2 8828.87} C_VEL
LIN {X 0,Y 589.526,Z 1224.941,A -85,B 0,C 180,E1 8832.42,E2 8832.42} C_VEL
LIN {X 0,Y 590.932,Z 1204.146,A -85,B 0,C 180,E1 8835.995,E2 8835.995} C_VEL
LIN {X 0,Y 592.776,Z 1179.651,A -85,B 0,C 180,E1 8839.096,E2 8839.096} C_VEL
LIN {X 0,Y 595.208,Z 1149.981,A -85,B 0,C 180,E1 8841.918,E2 8841.918} C_VEL
LIN {X 0,Y 597.57,Z 1118.173,A -85,B 0,C 180,E1 8844.199,E2 8844.199} C_VEL
LIN {X 0,Y 600.09,Z 1081.115,A -85,B 0,C 180,E1 8846.141,E2 8846.141} C_VEL
LIN {X 0,Y 602.193,Z 1040.945,A -85,B 0,C 180,E1 8847.574,E2 8847.574} C_VEL
LIN {X 0,Y 602.151,Z 1020.821,A -85,B 0,C 180,E1 8848.096,E2 8848.096} C_VEL
LIN {X 0,Y 587.488,Z 977.53,A -85,B 0,C 180,E1 8849.657,E2 8849.657} C_VEL
LIN {X 0,Y 587.345,Z 977.53,A -85,B 0,C 180,E1 8854.563,E2 8854.563} C_VEL
LIN {X 0,Y 587.162,Z 977.53,A -85,B 0,C 180,E1 8860.528,E2 8860.528} C_VEL
LIN {X 0,Y 587.14,Z 977.53,A -85,B 0,C 180,E1 8863.843,E2 8863.843} C_VEL
LIN {X 0,Y 583.218,Z 977.53,A -85,B 0,C 180,E1 8865.499,E2 8865.499} C_VEL
LIN {X 0,Y 579.176,Z 977.53,A -85,B 0,C 180,E1 8867.179,E2 8867.179} C_VEL
LIN {X 0,Y 579.433,Z 977.53,A -85,B 0,C 180,E1 8873.034,E2 8873.034} C_VEL
LIN {X 0,Y 579.498,Z 978.098,A -85,B 0,C 180,E1 8877.695,E2 8877.695} C_VEL
LIN {X 0,Y 589.465,Z 1019.662,A -85,B 0,C 180,E1 8880.518,E2 8880.518} C_VEL
LIN {X 0,Y 595.958,Z 1034.569,A -85,B 0,C 180,E1 8880.997,E2 8880.997} C_VEL
LIN {X 0,Y 594.652,Z 1079.197,A -85,B 0,C 180,E1 8881.775,E2 8881.775} C_VEL
LIN {X 0,Y 592.584,Z 1118.044,A -85,B 0,C 180,E1 8882.99,E2 8882.99} C_VEL
LIN {X 0,Y 589.986,Z 1155.48,A -85,B 0,C 180,E1 8884.732,E2 8884.732} C_VEL
LIN {X 0,Y 587.447,Z 1190.596,A -85,B 0,C 180,E1 8886.991,E2 8886.991} C_VEL
LIN {X 0,Y 585.064,Z 1222.689,A -85,B 0,C 180,E1 8889.74,E2 8889.74} C_VEL
LIN {X 0,Y 583.021,Z 1251.156,A -85,B 0,C 180,E1 8893.006,E2 8893.006} C_VEL
LIN {X 0,Y 581.688,Z 1273.599,A -85,B 0,C 180,E1 8896.448,E2 8896.448} C_VEL
LIN {X 0,Y 580.952,Z 1291.227,A -85,B 0,C 180,E1 8900.246,E2 8900.246} C_VEL
LIN {X 0,Y 580.649,Z 1302.568,A -85,B 0,C 180,E1 8904.015,E2 8904.015} C_VEL
LIN {X 0,Y 580.64,Z 1307.601,A -85,B 0,C 180,E1 8907.015,E2 8907.015} C_VEL
LIN {X 0,Y 580.646,Z 1309.218,A -85,B 0,C 180,E1 8910.007,E2 8910.007} C_VEL
LIN {X 0,Y 580.627,Z 1306.464,A -85,B 0,C 180,E1 8913.748,E2 8913.748} C_VEL
LIN {X 0,Y 580.831,Z 1298.244,A -85,B 0,C 180,E1 8917.678,E2 8917.678} C_VEL
LIN {X 0,Y 581.273,Z 1283.533,A -85,B 0,C 180,E1 8921.663,E2 8921.663} C_VEL
LIN {X 0,Y 582.257,Z 1263.988,A -85,B 0,C 180,E1 8925.268,E2 8925.268} C_VEL
LIN {X 0,Y 583.895,Z 1240.117,A -85,B 0,C 180,E1 8928.515,E2 8928.515} C_VEL
LIN {X 0,Y 586.212,Z 1210.744,A -85,B 0,C 180,E1 8931.527,E2 8931.527} C_VEL
LIN {X 0,Y 588.943,Z 1177.416,A -85,B 0,C 180,E1 8934.093,E2 8934.093} C_VEL
LIN {X 0,Y 591.657,Z 1141.457,A -85,B 0,C 180,E1 8936.136,E2 8936.136} C_VEL
LIN {X 0,Y 594.151,Z 1101.386,A -85,B 0,C 180,E1 8937.718,E2 8937.718} C_VEL
LIN {X 0,Y 595.865,Z 1060.5,A -85,B 0,C 180,E1 8938.692,E2 8938.692} C_VEL
LIN {X 0,Y 595.537,Z 1031.99,A -85,B 0,C 180,E1 8939.139,E2 8939.139} C_VEL
LIN {X 0,Y 585.647,Z 1004.768,A -85,B 0,C 180,E1 8940.006,E2 8940.006} C_VEL
LIN {X 0,Y 579.547,Z 977.53,A -85,B 0,C 180,E1 8941.824,E2 8941.824} C_VEL
LIN {X 0,Y 579.4,Z 977.53,A -85,B 0,C 180,E1 8946.986,E2 8946.986} C_VEL
LIN {X 0,Y 579.378,Z 977.53,A -85,B 0,C 180,E1 8952.944,E2 8952.944} C_VEL
LIN {X 0,Y 579.328,Z 977.53,A -85,B 0,C 180,E1 8959.185,E2 8959.185} C_VEL
LIN {X 0,Y 579.305,Z 977.53,A -85,B 0,C 180,E1 8964.887,E2 8964.887} C_VEL
LIN {X 0,Y 579.48,Z 977.53,A -85,B 0,C 180,E1 8970.226,E2 8970.226} C_VEL
LIN {X 0,Y 579.659,Z 977.53,A -85,B 0,C 180,E1 8975.291,E2 8975.291} C_VEL
LIN {X 0,Y 579.781,Z 977.53,A -85,B 0,C 180,E1 8980.217,E2 8980.217} C_VEL
LIN {X 0,Y 579.817,Z 977.53,A -85,B 0,C 180,E1 8985.253,E2 8985.253} C_VEL
LIN {X 0,Y 580.008,Z 977.53,A -85,B 0,C 180,E1 8990.994,E2 8990.994} C_VEL
LIN {X 0,Y 580.101,Z 977.53,A -85,B 0,C 180,E1 8992.293,E2 8992.293} C_VEL
LIN {X 0,Y 589.309,Z 1008.079,A -85,B 0,C 180,E1 8993.425,E2 8993.425} C_VEL
LIN {X 0,Y 587.751,Z 1065.011,A -85,B 0,C 180,E1 8994.649,E2 8994.649} C_VEL
LIN {X 0,Y 586.72,Z 1093.225,A -85,B 0,C 180,E1 8995.846,E2 8995.846} C_VEL
LIN {X 0,Y 585.303,Z 1118.922,A -85,B 0,C 180,E1 8997.6,E2 8997.6} C_VEL
LIN {X 0,Y 583.889,Z 1140.737,A -85,B 0,C 180,E1 8999.825,E2 8999.825} C_VEL
LIN {X 0,Y 582.79,Z 1156.741,A -85,B 0,C 180,E1 9002.245,E2 9002.245} C_VEL
LIN {X 0,Y 581.957,Z 1167.888,A -85,B 0,C 180,E1 9004.864,E2 9004.864} C_VEL
LIN {X 0,Y 581.451,Z 1174.533,A -85,B 0,C 180,E1 9007.945,E2 9007.945} C_VEL
LIN {X 0,Y 581.344,Z 1175.234,A -85,B 0,C 180,E1 9010.522,E2 9010.522} C_VEL
LIN {X 0,Y 581.528,Z 1170.453,A -85,B 0,C 180,E1 9013.572,E2 9013.572} C_VEL
LIN {X 0,Y 581.959,Z 1160.548,A -85,B 0,C 180,E1 9016.323,E2 9016.323} C_VEL
LIN {X 0,Y 582.744,Z 1144.877,A -85,B 0,C 180,E1 9018.976,E2 9018.976} C_VEL
LIN {X 0,Y 583.828,Z 1123.929,A -85,B 0,C 180,E1 9021.315,E2 9021.315} C_VEL
LIN {X 0,Y 584.988,Z 1099.351,A -85,B 0,C 180,E1 9023.176,E2 9023.176} C_VEL
LIN {X 0,Y 586.067,Z 1071.199,A -85,B 0,C 180,E1 9024.551,E2 9024.551} C_VEL
LIN {X 0,Y 586.601,Z 1042.016,A -85,B 0,C 180,E1 9025.348,E2 9025.348} C_VEL
LIN {X 0,Y 586.664,Z 1003.436,A -85,B 0,C 180,E1 9025.976,E2 9025.976} C_VEL
LIN {X 0,Y 579.764,Z 977.53,A -85,B 0,C 180,E1 9026.7,E2 9026.7} C_VEL
LIN {X 0,Y 579.49,Z 977.53,A -85,B 0,C 180,E1 9033.19,E2 9033.19} C_VEL
LIN {X 0,Y 579.359,Z 977.53,A -85,B 0,C 180,E1 9038.889,E2 9038.889} C_VEL
LIN {X 0,Y 579.371,Z 977.53,A -85,B 0,C 180,E1 9045.068,E2 9045.068} C_VEL
LIN {X 0,Y 579.297,Z 977.53,A -85,B 0,C 180,E1 9051.106,E2 9051.106} C_VEL
LIN {X 0,Y 579.401,Z 977.53,A -85,B 0,C 180,E1 9056.82,E2 9056.82} C_VEL
LIN {X 0,Y 579.583,Z 977.53,A -85,B 0,C 180,E1 9062.745,E2 9062.745} C_VEL
LIN {X 0,Y 579.7,Z 977.53,A -85,B 0,C 180,E1 9068.527,E2 9068.527} C_VEL
LIN {X 0,Y 579.811,Z 977.53,A -85,B 0,C 180,E1 9073.286,E2 9073.286} C_VEL
LIN {X 0,Y 579.96,Z 977.53,A -85,B 0,C 180,E1 9079.455,E2 9079.455} C_VEL
LIN {X 0,Y 580.134,Z 977.53,A -85,B 0,C 180,E1 9083.996,E2 9083.996} C_VEL
LIN {X 0,Y 580.232,Z 977.53,A -85,B 0,C 180,E1 9088.497,E2 9088.497} C_VEL
LIN {X 0,Y 580.225,Z 977.53,A -85,B 0,C 180,E1 9092.987,E2 9092.987} C_VEL
LIN {X 0,Y 580.005,Z 977.53,A -85,B 0,C 180,E1 9097.499,E2 9097.499} C_VEL
LIN {X 0,Y 579.916,Z 977.53,A -85,B 0,C 180,E1 9102.058,E2 9102.058} C_VEL
LIN {X 0,Y 579.824,Z 977.53,A -85,B 0,C 180,E1 9106.699,E2 9106.699} C_VEL
LIN {X 0,Y 579.678,Z 977.53,A -85,B 0,C 180,E1 9111.459,E2 9111.459} C_VEL
LIN {X 0,Y 579.547,Z 977.53,A -85,B 0,C 180,E1 9117.248,E2 9117.248} C_VEL
LIN {X 0,Y 579.431,Z 977.53,A -85,B 0,C 180,E1 9123.302,E2 9123.302} C_VEL
LIN {X 0,Y 579.353,Z 977.53,A -85,B 0,C 180,E1 9128.872,E2 9128.872} C_VEL
LIN {X 0,Y 579.349,Z 977.53,A -85,B 0,C 180,E1 9135.067,E2 9135.067} C_VEL
LIN {X 0,Y 579.299,Z 977.53,A -85,B 0,C 180,E1 9141.106,E2 9141.106} C_VEL
LIN {X 0,Y 579.413,Z 977.53,A -85,B 0,C 180,E1 9146.797,E2 9146.797} C_VEL
LIN {X 0,Y 579.563,Z 977.559,A -85,B 0,C 180,E1 9149.779,E2 9149.779} C_VEL
LIN {X 0,Y 596.457,Z 1024.358,A -85,B 0,C 180,E1 9151.417,E2 9151.417} C_VEL
LIN {X 0,Y 594.415,Z 1065.549,A -85,B 0,C 180,E1 9152.679,E2 9152.679} C_VEL
LIN {X 0,Y 591.851,Z 1102.413,A -85,B 0,C 180,E1 9154.395,E2 9154.395} C_VEL
LIN {X 0,Y 589.041,Z 1136.472,A -85,B 0,C 180,E1 9156.593,E2 9156.593} C_VEL
LIN {X 0,Y 586.392,Z 1166.567,A -85,B 0,C 180,E1 9159.179,E2 9159.179} C_VEL
LIN {X 0,Y 584,Z 1193.59,A -85,B 0,C 180,E1 9162.241,E2 9162.241} C_VEL
LIN {X 0,Y 582.281,Z 1216.244,A -85,B 0,C 180,E1 9165.678,E2 9165.678} C_VEL
LIN {X 0,Y 581.241,Z 1232.689,A -85,B 0,C 180,E1 9169.096,E2 9169.096} C_VEL
LIN {X 0,Y 580.755,Z 1244.081,A -85,B 0,C 180,E1 9172.494,E2 9172.494} C_VEL
LIN {X 0,Y 580.49,Z 1250.433,A -85,B 0,C 180,E1 9175.498,E2 9175.498} C_VEL
LIN {X 0,Y 580.467,Z 1253.61,A -85,B 0,C 180,E1 9178.494,E2 9178.494} C_VEL
LIN {X 0,Y 580.603,Z 1253.601,A -85,B 0,C 180,E1 9181.485,E2 9181.485} C_VEL
LIN {X 0,Y 580.67,Z 1249.227,A -85,B 0,C 180,E1 9185.229,E2 9185.229} C_VEL
LIN {X 0,Y 580.979,Z 1239.672,A -85,B 0,C 180,E1 9188.991,E2 9188.991} C_VEL
LIN {X 0,Y 581.831,Z 1223.975,A -85,B 0,C 180,E1 9192.826,E2 9192.826} C_VEL
LIN {X 0,Y 583.219,Z 1204.301,A -85,B 0,C 180,E1 9196.208,E2 9196.208} C_VEL
LIN {X 0,Y 585.17,Z 1179.662,A -85,B 0,C 180,E1 9199.355,E2 9199.355} C_VEL
LIN {X 0,Y 587.686,Z 1150.483,A -85,B 0,C 180,E1 9202.16,E2 9202.16} C_VEL
LIN {X 0,Y 590.276,Z 1117.884,A -85,B 0,C 180,E1 9204.518,E2 9204.518} C_VEL
LIN {X 0,Y 592.823,Z 1081.899,A -85,B 0,C 180,E1 9206.425,E2 9206.425} C_VEL
LIN {X 0,Y 595.037,Z 1041.443,A -85,B 0,C 180,E1 9207.893,E2 9207.893} C_VEL
LIN {X 0,Y 595.062,Z 1023.094,A -85,B 0,C 180,E1 9208.383,E2 9208.383} C_VEL
LIN {X 0,Y 581.712,Z 984,A -85,B 0,C 180,E1 9209.811,E2 9209.811} C_VEL
LIN {X 0,Y 579.565,Z 977.53,A -85,B 0,C 180,E1 9210.096,E2 9210.096} C_VEL
LIN {X 0,Y 579.365,Z 977.53,A -85,B 0,C 180,E1 9215.841,E2 9215.841} C_VEL
LIN {X 0,Y 579.247,Z 977.53,A -85,B 0,C 180,E1 9220.822,E2 9220.822} C_VEL
LIN {X 0,Y 579.176,Z 977.53,A -85,B 0,C 180,E1 9227.179,E2 9227.179} C_VEL
LIN {X 0,Y 575.235,Z 977.53,A -85,B 0,C 180,E1 9228.862,E2 9228.862} C_VEL
LIN {X 0,Y 571.331,Z 977.53,A -85,B 0,C 180,E1 9230.569,E2 9230.569} C_VEL
LIN {X 0,Y 571.489,Z 977.53,A -85,B 0,C 180,E1 9236.174,E2 9236.174} C_VEL
LIN {X 0,Y 571.627,Z 977.812,A -85,B 0,C 180,E1 9237.322,E2 9237.322} C_VEL
LIN {X 0,Y 581.205,Z 1018.511,A -85,B 0,C 180,E1 9240.143,E2 9240.143} C_VEL
LIN {X 0,Y 588.675,Z 1037.123,A -85,B 0,C 180,E1 9240.729,E2 9240.729} C_VEL
LIN {X 0,Y 587.232,Z 1080.991,A -85,B 0,C 180,E1 9241.53,E2 9241.53} C_VEL
LIN {X 0,Y 584.922,Z 1122.832,A -85,B 0,C 180,E1 9242.913,E2 9242.913} C_VEL
LIN {X 0,Y 582.051,Z 1162.169,A -85,B 0,C 180,E1 9244.878,E2 9244.878} C_VEL
LIN {X 0,Y 579.11,Z 1198.436,A -85,B 0,C 180,E1 9247.407,E2 9247.407} C_VEL
LIN {X 0,Y 576.631,Z 1229.923,A -85,B 0,C 180,E1 9250.355,E2 9250.355} C_VEL
LIN {X 0,Y 574.738,Z 1255.974,A -85,B 0,C 180,E1 9253.588,E2 9253.588} C_VEL
LIN {X 0,Y 573.514,Z 1277.819,A -85,B 0,C 180,E1 9257.243,E2 9257.243} C_VEL
LIN {X 0,Y 572.947,Z 1293.213,A -85,B 0,C 180,E1 9260.877,E2 9260.877} C_VEL
LIN {X 0,Y 572.837,Z 1303.457,A -85,B 0,C 180,E1 9264.695,E2 9264.695} C_VEL
LIN {X 0,Y 572.804,Z 1308.207,A -85,B 0,C 180,E1 9268.491,E2 9268.491} C_VEL
LIN {X 0,Y 572.802,Z 1308.255,A -85,B 0,C 180,E1 9271.523,E2 9271.523} C_VEL
LIN {X 0,Y 572.824,Z 1303.671,A -85,B 0,C 180,E1 9275.319,E2 9275.319} C_VEL
LIN {X 0,Y 572.938,Z 1293.646,A -85,B 0,C 180,E1 9279.138,E2 9279.138} C_VEL
LIN {X 0,Y 573.645,Z 1277.96,A -85,B 0,C 180,E1 9282.904,E2 9282.904} C_VEL
LIN {X 0,Y 574.862,Z 1257.2,A -85,B 0,C 180,E1 9286.435,E2 9286.435} C_VEL
LIN {X 0,Y 576.829,Z 1231.769,A -85,B 0,C 180,E1 9289.653,E2 9289.653} C_VEL
LIN {X 0,Y 579.385,Z 1202.137,A -85,B 0,C 180,E1 9292.495,E2 9292.495} C_VEL
LIN {X 0,Y 582.176,Z 1168.5,A -85,B 0,C 180,E1 9294.926,E2 9294.926} C_VEL
LIN {X 0,Y 584.971,Z 1132.202,A -85,B 0,C 180,E1 9296.846,E2 9296.846} C_VEL
LIN {X 0,Y 587.329,Z 1093.283,A -85,B 0,C 180,E1 9298.263,E2 9298.263} C_VEL
LIN {X 0,Y 588.863,Z 1054.229,A -85,B 0,C 180,E1 9299.115,E2 9299.115} C_VEL
LIN {X 0,Y 588.458,Z 1034.509,A -85,B 0,C 180,E1 9299.432,E2 9299.432} C_VEL
LIN {X 0,Y 578.266,Z 1005.462,A -85,B 0,C 180,E1 9300.354,E2 9300.354} C_VEL
LIN {X 0,Y 576.017,Z 996.208,A -85,B 0,C 180,E1 9300.842,E2 9300.842} C_VEL
LIN {X 0,Y 571.618,Z 977.53,A -85,B 0,C 180,E1 9302.237,E2 9302.237} C_VEL
LIN {X 0,Y 571.476,Z 977.53,A -85,B 0,C 180,E1 9307.587,E2 9307.587} C_VEL
LIN {X 0,Y 571.417,Z 977.53,A -85,B 0,C 180,E1 9313.597,E2 9313.597} C_VEL
LIN {X 0,Y 571.346,Z 977.53,A -85,B 0,C 180,E1 9318.49,E2 9318.49} C_VEL
LIN {X 0,Y 571.401,Z 977.53,A -85,B 0,C 180,E1 9324.328,E2 9324.328} C_VEL
LIN {X 0,Y 571.589,Z 977.53,A -85,B 0,C 180,E1 9329.772,E2 9329.772} C_VEL
LIN {X 0,Y 571.712,Z 977.53,A -85,B 0,C 180,E1 9334.924,E2 9334.924} C_VEL
LIN {X 0,Y 571.827,Z 977.53,A -85,B 0,C 180,E1 9339.864,E2 9339.864} C_VEL
LIN {X 0,Y 571.897,Z 977.53,A -85,B 0,C 180,E1 9344.649,E2 9344.649} C_VEL
LIN {X 0,Y 572.01,Z 977.53,A -85,B 0,C 180,E1 9349.326,E2 9349.326} C_VEL
LIN {X 0,Y 572.161,Z 977.53,A -85,B 0,C 180,E1 9351.876,E2 9351.876} C_VEL
LIN {X 0,Y 582.057,Z 1010.244,A -85,B 0,C 180,E1 9353.142,E2 9353.142} C_VEL
LIN {X 0,Y 580.409,Z 1066.233,A -85,B 0,C 180,E1 9354.393,E2 9354.393} C_VEL
LIN {X 0,Y 579.279,Z 1094.196,A -85,B 0,C 180,E1 9355.604,E2 9355.604} C_VEL
LIN {X 0,Y 577.778,Z 1119.851,A -85,B 0,C 180,E1 9357.381,E2 9357.381} C_VEL
LIN {X 0,Y 576.28,Z 1141.562,A -85,B 0,C 180,E1 9359.619,E2 9359.619} C_VEL
LIN {X 0,Y 575,Z 1158.619,A -85,B 0,C 180,E1 9362.276,E2 9362.276} C_VEL
LIN {X 0,Y 574.137,Z 1169.404,A -85,B 0,C 180,E1 9364.931,E2 9364.931} C_VEL
LIN {X 0,Y 573.652,Z 1175.137,A -85,B 0,C 180,E1 9367.599,E2 9367.599} C_VEL
LIN {X 0,Y 573.514,Z 1176.096,A -85,B 0,C 180,E1 9370.668,E2 9370.668} C_VEL
LIN {X 0,Y 573.7,Z 1170.947,A -85,B 0,C 180,E1 9373.761,E2 9373.761} C_VEL
LIN {X 0,Y 574.156,Z 1160.972,A -85,B 0,C 180,E1 9376.491,E2 9376.491} C_VEL
LIN {X 0,Y 574.966,Z 1145.99,A -85,B 0,C 180,E1 9379.043,E2 9379.043} C_VEL
LIN {X 0,Y 576.114,Z 1124.788,A -85,B 0,C 180,E1 9381.449,E2 9381.449} C_VEL
LIN {X 0,Y 577.303,Z 1100.995,A -85,B 0,C 180,E1 9383.286,E2 9383.286} C_VEL
LIN {X 0,Y 578.42,Z 1073.344,A -85,B 0,C 180,E1 9384.686,E2 9384.686} C_VEL
LIN {X 0,Y 578.991,Z 1044.355,A -85,B 0,C 180,E1 9385.521,E2 9385.521} C_VEL
LIN {X 0,Y 578.877,Z 1003.897,A -85,B 0,C 180,E1 9386.209,E2 9386.209} C_VEL
LIN {X 0,Y 571.832,Z 977.53,A -85,B 0,C 180,E1 9386.936,E2 9386.936} C_VEL
LIN {X 0,Y 571.557,Z 977.53,A -85,B 0,C 180,E1 9392.029,E2 9392.029} C_VEL
LIN {X 0,Y 571.445,Z 977.53,A -85,B 0,C 180,E1 9397.589,E2 9397.589} C_VEL
LIN {X 0,Y 571.415,Z 977.53,A -85,B 0,C 180,E1 9403.596,E2 9403.596} C_VEL
LIN {X 0,Y 571.351,Z 977.53,A -85,B 0,C 180,E1 9408.46,E2 9408.46} C_VEL
LIN {X 0,Y 571.408,Z 977.53,A -85,B 0,C 180,E1 9414.302,E2 9414.302} C_VEL
LIN {X 0,Y 571.558,Z 977.53,A -85,B 0,C 180,E1 9419.746,E2 9419.746} C_VEL
LIN {X 0,Y 571.694,Z 977.53,A -85,B 0,C 180,E1 9424.9,E2 9424.9} C_VEL
LIN {X 0,Y 571.812,Z 977.53,A -85,B 0,C 180,E1 9429.842,E2 9429.842} C_VEL
LIN {X 0,Y 571.922,Z 977.53,A -85,B 0,C 180,E1 9434.629,E2 9434.629} C_VEL
LIN {X 0,Y 572.04,Z 977.53,A -85,B 0,C 180,E1 9439.307,E2 9439.307} C_VEL
LIN {X 0,Y 572.236,Z 977.53,A -85,B 0,C 180,E1 9443.913,E2 9443.913} C_VEL
LIN {X 0,Y 572.33,Z 977.53,A -85,B 0,C 180,E1 9448.476,E2 9448.476} C_VEL
LIN {X 0,Y 572.326,Z 977.53,A -85,B 0,C 180,E1 9453.028,E2 9453.028} C_VEL
LIN {X 0,Y 572.092,Z 977.53,A -85,B 0,C 180,E1 9457.603,E2 9457.603} C_VEL
LIN {X 0,Y 571.998,Z 977.53,A -85,B 0,C 180,E1 9462.228,E2 9462.228} C_VEL
LIN {X 0,Y 571.874,Z 977.53,A -85,B 0,C 180,E1 9467.456,E2 9467.456} C_VEL
LIN {X 0,Y 571.71,Z 977.53,A -85,B 0,C 180,E1 9473.418,E2 9473.418} C_VEL
LIN {X 0,Y 571.567,Z 977.53,A -85,B 0,C 180,E1 9478.962,E2 9478.962} C_VEL
LIN {X 0,Y 571.446,Z 977.53,A -85,B 0,C 180,E1 9484.705,E2 9484.705} C_VEL
LIN {X 0,Y 571.398,Z 977.53,A -85,B 0,C 180,E1 9489.724,E2 9489.724} C_VEL
LIN {X 0,Y 571.364,Z 977.53,A -85,B 0,C 180,E1 9495.718,E2 9495.718} C_VEL
LIN {X 0,Y 571.345,Z 977.53,A -85,B 0,C 180,E1 9500.46,E2 9500.46} C_VEL
LIN {X 0,Y 571.41,Z 977.53,A -85,B 0,C 180,E1 9506.151,E2 9506.151} C_VEL
LIN {X 0,Y 571.643,Z 977.954,A -85,B 0,C 180,E1 9509.39,E2 9509.39} C_VEL
LIN {X 0,Y 589.022,Z 1025.555,A -85,B 0,C 180,E1 9511.103,E2 9511.103} C_VEL
LIN {X 0,Y 587.085,Z 1067.135,A -85,B 0,C 180,E1 9512.424,E2 9512.424} C_VEL
LIN {X 0,Y 584.446,Z 1103.463,A -85,B 0,C 180,E1 9514.15,E2 9514.15} C_VEL
LIN {X 0,Y 581.452,Z 1138.165,A -85,B 0,C 180,E1 9516.432,E2 9516.432} C_VEL
LIN {X 0,Y 578.703,Z 1168.342,A -85,B 0,C 180,E1 9519.09,E2 9519.09} C_VEL
LIN {X 0,Y 576.214,Z 1195.051,A -85,B 0,C 180,E1 9522.191,E2 9522.191} C_VEL
LIN {X 0,Y 574.444,Z 1217.46,A -85,B 0,C 180,E1 9525.673,E2 9525.673} C_VEL
LIN {X 0,Y 573.344,Z 1234.444,A -85,B 0,C 180,E1 9529.329,E2 9529.329} C_VEL
LIN {X 0,Y 572.832,Z 1246.535,A -85,B 0,C 180,E1 9533.249,E2 9533.249} C_VEL
LIN {X 0,Y 572.622,Z 1252.761,A -85,B 0,C 180,E1 9536.956,E2 9536.956} C_VEL
LIN {X 0,Y 572.645,Z 1254.397,A -85,B 0,C 180,E1 9539.989,E2 9539.989} C_VEL
LIN {X 0,Y 572.685,Z 1252.792,A -85,B 0,C 180,E1 9543.022,E2 9543.022} C_VEL
LIN {X 0,Y 572.861,Z 1246.549,A -85,B 0,C 180,E1 9546.75,E2 9546.75} C_VEL
LIN {X 0,Y 573.397,Z 1234.51,A -85,B 0,C 180,E1 9550.648,E2 9550.648} C_VEL
LIN {X 0,Y 574.447,Z 1217.442,A -85,B 0,C 180,E1 9554.304,E2 9554.304} C_VEL
LIN {X 0,Y 576.153,Z 1196.281,A -85,B 0,C 180,E1 9557.591,E2 9557.591} C_VEL
LIN {X 0,Y 578.572,Z 1169.615,A -85,B 0,C 180,E1 9560.691,E2 9560.691} C_VEL
LIN {X 0,Y 581.299,Z 1138.985,A -85,B 0,C 180,E1 9563.373,E2 9563.373} C_VEL
LIN {X 0,Y 584.106,Z 1104.276,A -85,B 0,C 180,E1 9565.637,E2 9565.637} C_VEL
LIN {X 0,Y 586.736,Z 1065.394,A -85,B 0,C 180,E1 9567.442,E2 9567.442} C_VEL
LIN {X 0,Y 587.843,Z 1024.682,A -85,B 0,C 180,E1 9568.707,E2 9568.707} C_VEL
LIN {X 0,Y 575.324,Z 987.344,A -85,B 0,C 180,E1 9570.13,E2 9570.13} C_VEL
LIN {X 0,Y 571.619,Z 977.53,A -85,B 0,C 180,E1 9570.557,E2 9570.557} C_VEL
LIN {X 0,Y 571.467,Z 977.53,A -85,B 0,C 180,E1 9575.667,E2 9575.667} C_VEL
LIN {X 0,Y 571.245,Z 977.53,A -85,B 0,C 180,E1 9581.519,E2 9581.519} C_VEL
LIN {X 0,Y 571.175,Z 977.53,A -85,B 0,C 180,E1 9587.18,E2 9587.18} C_VEL
LIN {X 0,Y 571.331,Z 977.53,A -85,B 0,C 180,E1 9590.569,E2 9590.569} C_VEL
LIN {X 0,Y 567.447,Z 977.53,A -85,B 0,C 180,E1 9592.275,E2 9592.275} C_VEL
LIN {X 0,Y 563.526,Z 977.53,A -85,B 0,C 180,E1 9594.004,E2 9594.004} C_VEL
LIN {X 0,Y 563.715,Z 978.264,A -85,B 0,C 180,E1 9596.986,E2 9596.986} C_VEL
LIN {X 0,Y 573.096,Z 1017.046,A -85,B 0,C 180,E1 9599.708,E2 9599.708} C_VEL
LIN {X 0,Y 581.388,Z 1040.299,A -85,B 0,C 180,E1 9600.465,E2 9600.465} C_VEL
LIN {X 0,Y 579.743,Z 1085.117,A -85,B 0,C 180,E1 9601.351,E2 9601.351} C_VEL
LIN {X 0,Y 577.175,Z 1126.342,A -85,B 0,C 180,E1 9602.804,E2 9602.804} C_VEL
LIN {X 0,Y 574.371,Z 1163.419,A -85,B 0,C 180,E1 9604.728,E2 9604.728} C_VEL
LIN {X 0,Y 571.447,Z 1198.062,A -85,B 0,C 180,E1 9607.19,E2 9607.19} C_VEL
LIN {X 0,Y 568.862,Z 1229.675,A -85,B 0,C 180,E1 9610.198,E2 9610.198} C_VEL
LIN {X 0,Y 566.821,Z 1257.139,A -85,B 0,C 180,E1 9613.647,E2 9613.647} C_VEL
LIN {X 0,Y 565.618,Z 1278.086,A -85,B 0,C 180,E1 9617.239,E2 9617.239} C_VEL
LIN {X 0,Y 565.056,Z 1293.969,A -85,B 0,C 180,E1 9621.137,E2 9621.137} C_VEL
LIN {X 0,Y 564.946,Z 1303.045,A -85,B 0,C 180,E1 9624.621,E2 9624.621} C_VEL
LIN {X 0,Y 564.909,Z 1307.825,A -85,B 0,C 180,E1 9628.47,E2 9628.47} C_VEL
LIN {X 0,Y 564.907,Z 1307.882,A -85,B 0,C 180,E1 9631.544,E2 9631.544} C_VEL
LIN {X 0,Y 564.941,Z 1303.283,A -85,B 0,C 180,E1 9635.394,E2 9635.394} C_VEL
LIN {X 0,Y 565.05,Z 1293.215,A -85,B 0,C 180,E1 9639.266,E2 9639.266} C_VEL
LIN {X 0,Y 565.821,Z 1277.05,A -85,B 0,C 180,E1 9643.165,E2 9643.165} C_VEL
LIN {X 0,Y 567.131,Z 1256.091,A -85,B 0,C 180,E1 9646.738,E2 9646.738} C_VEL
LIN {X 0,Y 569.201,Z 1230.737,A -85,B 0,C 180,E1 9649.96,E2 9649.96} C_VEL
LIN {X 0,Y 571.982,Z 1199.994,A -85,B 0,C 180,E1 9652.906,E2 9652.906} C_VEL
LIN {X 0,Y 574.906,Z 1165.732,A -85,B 0,C 180,E1 9655.367,E2 9655.367} C_VEL
LIN {X 0,Y 577.913,Z 1127.944,A -85,B 0,C 180,E1 9657.334,E2 9657.334} C_VEL
LIN {X 0,Y 580.422,Z 1087.102,A -85,B 0,C 180,E1 9658.757,E2 9658.757} C_VEL
LIN {X 0,Y 581.855,Z 1044.013,A -85,B 0,C 180,E1 9659.601,E2 9659.601} C_VEL
LIN {X 0,Y 580.668,Z 1035.321,A -85,B 0,C 180,E1 9659.787,E2 9659.787} C_VEL
LIN {X 0,Y 568.859,Z 999.105,A -85,B 0,C 180,E1 9661.001,E2 9661.001} C_VEL
LIN {X 0,Y 563.661,Z 977.53,A -85,B 0,C 180,E1 9662.661,E2 9662.661} C_VEL
LIN {X 0,Y 563.458,Z 977.53,A -85,B 0,C 180,E1 9668.777,E2 9668.777} C_VEL
LIN {X 0,Y 563.505,Z 977.53,A -85,B 0,C 180,E1 9674.368,E2 9674.368} C_VEL
LIN {X 0,Y 563.407,Z 977.53,A -85,B 0,C 180,E1 9679.819,E2 9679.819} C_VEL
LIN {X 0,Y 563.479,Z 977.53,A -85,B 0,C 180,E1 9685.635,E2 9685.635} C_VEL
LIN {X 0,Y 563.691,Z 977.53,A -85,B 0,C 180,E1 9691.079,E2 9691.079} C_VEL
LIN {X 0,Y 563.817,Z 977.53,A -85,B 0,C 180,E1 9696.241,E2 9696.241} C_VEL
LIN {X 0,Y 563.928,Z 977.53,A -85,B 0,C 180,E1 9701.204,E2 9701.204} C_VEL
LIN {X 0,Y 563.968,Z 977.53,A -85,B 0,C 180,E1 9706.02,E2 9706.02} C_VEL
LIN {X 0,Y 564.267,Z 978.069,A -85,B 0,C 180,E1 9711.446,E2 9711.446} C_VEL
LIN {X 0,Y 574.911,Z 1011.116,A -85,B 0,C 180,E1 9712.824,E2 9712.824} C_VEL
LIN {X 0,Y 573.082,Z 1067.605,A -85,B 0,C 180,E1 9714.131,E2 9714.131} C_VEL
LIN {X 0,Y 571.865,Z 1095.314,A -85,B 0,C 180,E1 9715.357,E2 9715.357} C_VEL
LIN {X 0,Y 570.273,Z 1120.799,A -85,B 0,C 180,E1 9717.156,E2 9717.156} C_VEL
LIN {X 0,Y 568.694,Z 1141.968,A -85,B 0,C 180,E1 9719.357,E2 9719.357} C_VEL
LIN {X 0,Y 567.384,Z 1158.587,A -85,B 0,C 180,E1 9721.924,E2 9721.924} C_VEL
LIN {X 0,Y 566.431,Z 1169.735,A -85,B 0,C 180,E1 9724.614,E2 9724.614} C_VEL
LIN {X 0,Y 565.825,Z 1176.334,A -85,B 0,C 180,E1 9727.705,E2 9727.705} C_VEL
LIN {X 0,Y 565.665,Z 1176.91,A -85,B 0,C 180,E1 9730.817,E2 9730.817} C_VEL
LIN {X 0,Y 565.901,Z 1171.441,A -85,B 0,C 180,E1 9733.954,E2 9733.954} C_VEL
LIN {X 0,Y 566.454,Z 1160.119,A -85,B 0,C 180,E1 9736.922,E2 9736.922} C_VEL
LIN {X 0,Y 567.299,Z 1144.165,A -85,B 0,C 180,E1 9739.513,E2 9739.513} C_VEL
LIN {X 0,Y 568.552,Z 1123.566,A -85,B 0,C 180,E1 9741.782,E2 9741.782} C_VEL
LIN {X 0,Y 569.783,Z 1099.12,A -85,B 0,C 180,E1 9743.623,E2 9743.623} C_VEL
LIN {X 0,Y 570.899,Z 1070.009,A -85,B 0,C 180,E1 9745.033,E2 9745.033} C_VEL
LIN {X 0,Y 571.455,Z 1040.35,A -85,B 0,C 180,E1 9745.815,E2 9745.815} C_VEL
LIN {X 0,Y 571.307,Z 1005.128,A -85,B 0,C 180,E1 9746.427,E2 9746.427} C_VEL
LIN {X 0,Y 563.856,Z 977.53,A -85,B 0,C 180,E1 9747.193,E2 9747.193} C_VEL
LIN {X 0,Y 563.578,Z 977.53,A -85,B 0,C 180,E1 9752.538,E2 9752.538} C_VEL
LIN {X 0,Y 563.461,Z 977.53,A -85,B 0,C 180,E1 9758.217,E2 9758.217} C_VEL
LIN {X 0,Y 563.511,Z 977.53,A -85,B 0,C 180,E1 9763.436,E2 9763.436} C_VEL
LIN {X 0,Y 563.429,Z 977.53,A -85,B 0,C 180,E1 9768.862,E2 9768.862} C_VEL
LIN {X 0,Y 563.464,Z 977.53,A -85,B 0,C 180,E1 9773.79,E2 9773.79} C_VEL
LIN {X 0,Y 563.639,Z 977.53,A -85,B 0,C 180,E1 9779.358,E2 9779.358} C_VEL
LIN {X 0,Y 563.772,Z 977.53,A -85,B 0,C 180,E1 9784.522,E2 9784.522} C_VEL
LIN {X 0,Y 563.892,Z 977.53,A -85,B 0,C 180,E1 9790.15,E2 9790.15} C_VEL
LIN {X 0,Y 564.005,Z 977.53,A -85,B 0,C 180,E1 9796,E2 9796} C_VEL
LIN {X 0,Y 564.175,Z 977.53,A -85,B 0,C 180,E1 9800.719,E2 9800.719} C_VEL
LIN {X 0,Y 564.4,Z 977.53,A -85,B 0,C 180,E1 9805.373,E2 9805.373} C_VEL
LIN {X 0,Y 564.59,Z 977.53,A -85,B 0,C 180,E1 9811.531,E2 9811.531} C_VEL
LIN {X 0,Y 564.263,Z 977.53,A -85,B 0,C 180,E1 9816.452,E2 9816.452} C_VEL
LIN {X 0,Y 564.074,Z 977.53,A -85,B 0,C 180,E1 9822.402,E2 9822.402} C_VEL
LIN {X 0,Y 563.999,Z 977.53,A -85,B 0,C 180,E1 9827.182,E2 9827.182} C_VEL
LIN {X 0,Y 563.825,Z 977.53,A -85,B 0,C 180,E1 9832.094,E2 9832.094} C_VEL
LIN {X 0,Y 563.653,Z 977.53,A -85,B 0,C 180,E1 9837.474,E2 9837.474} C_VEL
LIN {X 0,Y 563.558,Z 977.53,A -85,B 0,C 180,E1 9842.522,E2 9842.522} C_VEL
LIN {X 0,Y 563.463,Z 977.53,A -85,B 0,C 180,E1 9848.199,E2 9848.199} C_VEL
LIN {X 0,Y 563.486,Z 977.53,A -85,B 0,C 180,E1 9853.435,E2 9853.435} C_VEL
LIN {X 0,Y 563.429,Z 977.53,A -85,B 0,C 180,E1 9858.842,E2 9858.842} C_VEL
LIN {X 0,Y 563.476,Z 977.53,A -85,B 0,C 180,E1 9863.766,E2 9863.766} C_VEL
LIN {X 0,Y 563.705,Z 977.53,A -85,B 0,C 180,E1 9868.966,E2 9868.966} C_VEL
LIN {X 0,Y 581.921,Z 1027.838,A -85,B 0,C 180,E1 9870.834,E2 9870.834} C_VEL
LIN {X 0,Y 579.904,Z 1066.942,A -85,B 0,C 180,E1 9872.092,E2 9872.092} C_VEL
LIN {X 0,Y 577.174,Z 1102.786,A -85,B 0,C 180,E1 9873.799,E2 9873.799} C_VEL
LIN {X 0,Y 574.116,Z 1137.488,A -85,B 0,C 180,E1 9876.092,E2 9876.092} C_VEL
LIN {X 0,Y 571.141,Z 1168.157,A -85,B 0,C 180,E1 9878.8,E2 9878.8} C_VEL
LIN {X 0,Y 568.539,Z 1195.048,A -85,B 0,C 180,E1 9881.942,E2 9881.942} C_VEL
LIN {X 0,Y 566.683,Z 1217.573,A -85,B 0,C 180,E1 9885.473,E2 9885.473} C_VEL
LIN {X 0,Y 565.514,Z 1234.662,A -85,B 0,C 180,E1 9889.18,E2 9889.18} C_VEL
LIN {X 0,Y 564.936,Z 1247.289,A -85,B 0,C 180,E1 9893.339,E2 9893.339} C_VEL
LIN {X 0,Y 564.728,Z 1253.113,A -85,B 0,C 180,E1 9896.913,E2 9896.913} C_VEL
LIN {X 0,Y 564.754,Z 1254.771,A -85,B 0,C 180,E1 9899.989,E2 9899.989} C_VEL
LIN {X 0,Y 564.793,Z 1253.169,A -85,B 0,C 180,E1 9903.064,E2 9903.064} C_VEL
LIN {X 0,Y 564.999,Z 1247.343,A -85,B 0,C 180,E1 9906.665,E2 9906.665} C_VEL
LIN {X 0,Y 565.474,Z 1236.333,A -85,B 0,C 180,E1 9910.408,E2 9910.408} C_VEL
LIN {X 0,Y 566.496,Z 1219.851,A -85,B 0,C 180,E1 9914.114,E2 9914.114} C_VEL
LIN {X 0,Y 568.385,Z 1197.916,A -85,B 0,C 180,E1 9917.639,E2 9917.639} C_VEL
LIN {X 0,Y 570.905,Z 1171.626,A -85,B 0,C 180,E1 9920.779,E2 9920.779} C_VEL
LIN {X 0,Y 573.76,Z 1141.558,A -85,B 0,C 180,E1 9923.488,E2 9923.488} C_VEL
LIN {X 0,Y 576.514,Z 1109.245,A -85,B 0,C 180,E1 9925.686,E2 9925.686} C_VEL
LIN {X 0,Y 579.203,Z 1072.115,A -85,B 0,C 180,E1 9927.524,E2 9927.524} C_VEL
LIN {X 0,Y 581.384,Z 1030.881,A -85,B 0,C 180,E1 9928.888,E2 9928.888} C_VEL
LIN {X 0,Y 571.596,Z 997.158,A -85,B 0,C 180,E1 9930.184,E2 9930.184} C_VEL
LIN {X 0,Y 563.699,Z 977.53,A -85,B 0,C 180,E1 9931.137,E2 9931.137} C_VEL
LIN {X 0,Y 563.528,Z 977.53,A -85,B 0,C 180,E1 9936.249,E2 9936.249} C_VEL
LIN {X 0,Y 563.339,Z 977.53,A -85,B 0,C 180,E1 9942.235,E2 9942.235} C_VEL
LIN {X 0,Y 563.333,Z 977.53,A -85,B 0,C 180,E1 9947.753,E2 9947.753} C_VEL
LIN {X 0,Y 563.56,Z 977.53,A -85,B 0,C 180,E1 9953.744,E2 9953.744} C_VEL
LIN {X 0,Y 563.526,Z 977.53,A -85,B 0,C 180,E1 9954.004,E2 9954.004} C_VEL
LIN {X 0,Y 559.552,Z 977.53,A -85,B 0,C 180,E1 9955.141,E2 9955.141} C_VEL
LIN {X 0,Y 555.706,Z 977.53,A -85,B 0,C 180,E1 9956.294,E2 9956.294} C_VEL
LIN {X 0,Y 555.787,Z 978.116,A -85,B 0,C 180,E1 9956.607,E2 9956.607} C_VEL
LIN {X 0,Y 564.209,Z 1012.623,A -85,B 0,C 180,E1 9959.08,E2 9959.08} C_VEL
LIN {X 0,Y 574.027,Z 1040.896,A -85,B 0,C 180,E1 9960.154,E2 9960.154} C_VEL
LIN {X 0,Y 572.442,Z 1084.416,A -85,B 0,C 180,E1 9961.04,E2 9961.04} C_VEL
LIN {X 0,Y 569.853,Z 1125.244,A -85,B 0,C 180,E1 9962.491,E2 9962.491} C_VEL
LIN {X 0,Y 566.824,Z 1163.032,A -85,B 0,C 180,E1 9964.473,E2 9964.473} C_VEL
LIN {X 0,Y 563.678,Z 1198.937,A -85,B 0,C 180,E1 9967.067,E2 9967.067} C_VEL
LIN {X 0,Y 561.112,Z 1230.279,A -85,B 0,C 180,E1 9970.074,E2 9970.074} C_VEL
LIN {X 0,Y 559.018,Z 1256.835,A -85,B 0,C 180,E1 9973.472,E2 9973.472} C_VEL
LIN {X 0,Y 557.794,Z 1277.509,A -85,B 0,C 180,E1 9977.057,E2 9977.057} C_VEL
LIN {X 0,Y 557.168,Z 1293.489,A -85,B 0,C 180,E1 9981.011,E2 9981.011} C_VEL
LIN {X 0,Y 557.039,Z 1302.617,A -85,B 0,C 180,E1 9984.544,E2 9984.544} C_VEL
LIN {X 0,Y 557.014,Z 1307.442,A -85,B 0,C 180,E1 9988.448,E2 9988.448} C_VEL
LIN {X 0,Y 557.011,Z 1307.509,A -85,B 0,C 180,E1 9991.566,E2 9991.566} C_VEL
LIN {X 0,Y 557.039,Z 1302.89,A -85,B 0,C 180,E1 9995.471,E2 9995.471} C_VEL
LIN {X 0,Y 557.174,Z 1292.771,A -85,B 0,C 180,E1 9999.398,E2 9999.398} C_VEL
LIN {X 0,Y 557.998,Z 1276.531,A -85,B 0,C 180,E1 10003.353,E2 10003.353} C_VEL
LIN {X 0,Y 559.384,Z 1255.72,A -85,B 0,C 180,E1 10006.937,E2 10006.937} C_VEL
LIN {X 0,Y 561.629,Z 1229.291,A -85,B 0,C 180,E1 10010.313,E2 10010.313} C_VEL
LIN {X 0,Y 564.434,Z 1199.011,A -85,B 0,C 180,E1 10013.23,E2 10013.23} C_VEL
LIN {X 0,Y 567.546,Z 1164.459,A -85,B 0,C 180,E1 10015.72,E2 10015.72} C_VEL
LIN {X 0,Y 570.762,Z 1125.435,A -85,B 0,C 180,E1 10017.745,E2 10017.745} C_VEL
LIN {X 0,Y 573.298,Z 1084.963,A -85,B 0,C 180,E1 10019.134,E2 10019.134} C_VEL
LIN {X 0,Y 574.771,Z 1042.682,A -85,B 0,C 180,E1 10019.957,E2 10019.957} C_VEL
LIN {X 0,Y 561.029,Z 998.965,A -85,B 0,C 180,E1 10021.392,E2 10021.392} C_VEL
LIN {X 0,Y 555.757,Z 977.53,A -85,B 0,C 180,E1 10023.116,E2 10023.116} C_VEL
LIN {X 0,Y 555.567,Z 977.53,A -85,B 0,C 180,E1 10028.861,E2 10028.861} C_VEL
LIN {X 0,Y 555.587,Z 977.53,A -85,B 0,C 180,E1 10034.861,E2 10034.861} C_VEL
LIN {X 0,Y 555.536,Z 977.53,A -85,B 0,C 180,E1 10039.804,E2 10039.804} C_VEL
LIN {X 0,Y 555.513,Z 977.53,A -85,B 0,C 180,E1 10045.072,E2 10045.072} C_VEL
LIN {X 0,Y 555.75,Z 977.53,A -85,B 0,C 180,E1 10050.763,E2 10050.763} C_VEL
LIN {X 0,Y 555.883,Z 977.53,A -85,B 0,C 180,E1 10055.881,E2 10055.881} C_VEL
LIN {X 0,Y 556.027,Z 977.53,A -85,B 0,C 180,E1 10060.926,E2 10060.926} C_VEL
LIN {X 0,Y 556.073,Z 977.53,A -85,B 0,C 180,E1 10065.817,E2 10065.817} C_VEL
LIN {X 0,Y 556.279,Z 977.53,A -85,B 0,C 180,E1 10070.947,E2 10070.947} C_VEL
LIN {X 0,Y 567.764,Z 1012.015,A -85,B 0,C 180,E1 10072.486,E2 10072.486} C_VEL
LIN {X 0,Y 565.751,Z 1069.064,A -85,B 0,C 180,E1 10073.862,E2 10073.862} C_VEL
LIN {X 0,Y 564.467,Z 1096.477,A -85,B 0,C 180,E1 10075.103,E2 10075.103} C_VEL
LIN {X 0,Y 562.81,Z 1121.845,A -85,B 0,C 180,E1 10076.925,E2 10076.925} C_VEL
LIN {X 0,Y 561.079,Z 1143.297,A -85,B 0,C 180,E1 10079.204,E2 10079.204} C_VEL
LIN {X 0,Y 559.607,Z 1160.502,A -85,B 0,C 180,E1 10081.95,E2 10081.95} C_VEL
LIN {X 0,Y 558.605,Z 1171.284,A -85,B 0,C 180,E1 10084.678,E2 10084.678} C_VEL
LIN {X 0,Y 557.98,Z 1177.511,A -85,B 0,C 180,E1 10087.814,E2 10087.814} C_VEL
LIN {X 0,Y 557.837,Z 1177.72,A -85,B 0,C 180,E1 10090.971,E2 10090.971} C_VEL
LIN {X 0,Y 558.083,Z 1171.914,A -85,B 0,C 180,E1 10094.154,E2 10094.154} C_VEL
LIN {X 0,Y 558.679,Z 1160.172,A -85,B 0,C 180,E1 10097.164,E2 10097.164} C_VEL
LIN {X 0,Y 559.617,Z 1143.803,A -85,B 0,C 180,E1 10099.792,E2 10099.792} C_VEL
LIN {X 0,Y 560.96,Z 1122.405,A -85,B 0,C 180,E1 10102.108,E2 10102.108} C_VEL
LIN {X 0,Y 562.249,Z 1097.271,A -85,B 0,C 180,E1 10103.959,E2 10103.959} C_VEL
LIN {X 0,Y 563.33,Z 1069.336,A -85,B 0,C 180,E1 10105.287,E2 10105.287} C_VEL
LIN {X 0,Y 563.988,Z 1037.207,A -85,B 0,C 180,E1 10106.095,E2 10106.095} C_VEL
LIN {X 0,Y 563.766,Z 1006.577,A -85,B 0,C 180,E1 10106.645,E2 10106.645} C_VEL
LIN {X 0,Y 555.929,Z 977.53,A -85,B 0,C 180,E1 10107.508,E2 10107.508} C_VEL
LIN {X 0,Y 555.645,Z 977.53,A -85,B 0,C 180,E1 10113.061,E2 10113.061} C_VEL
LIN {X 0,Y 555.575,Z 977.53,A -85,B 0,C 180,E1 10118.86,E2 10118.86} C_VEL
LIN {X 0,Y 555.584,Z 977.53,A -85,B 0,C 180,E1 10124.827,E2 10124.827} C_VEL
LIN {X 0,Y 555.523,Z 977.53,A -85,B 0,C 180,E1 10129.804,E2 10129.804} C_VEL
LIN {X 0,Y 555.531,Z 977.53,A -85,B 0,C 180,E1 10135.046,E2 10135.046} C_VEL
LIN {X 0,Y 555.722,Z 977.53,A -85,B 0,C 180,E1 10140.765,E2 10140.765} C_VEL
LIN {X 0,Y 555.873,Z 977.53,A -85,B 0,C 180,E1 10145.857,E2 10145.857} C_VEL
LIN {X 0,Y 556.006,Z 977.53,A -85,B 0,C 180,E1 10150.904,E2 10150.904} C_VEL
LIN {X 0,Y 556.107,Z 977.53,A -85,B 0,C 180,E1 10155.797,E2 10155.797} C_VEL
LIN {X 0,Y 556.257,Z 977.53,A -85,B 0,C 180,E1 10160.586,E2 10160.586} C_VEL
LIN {X 0,Y 556.493,Z 977.53,A -85,B 0,C 180,E1 10165.307,E2 10165.307} C_VEL
LIN {X 0,Y 556.683,Z 977.53,A -85,B 0,C 180,E1 10171.552,E2 10171.552} C_VEL
LIN {X 0,Y 556.415,Z 977.53,A -85,B 0,C 180,E1 10176.246,E2 10176.246} C_VEL
LIN {X 0,Y 556.18,Z 977.53,A -85,B 0,C 180,E1 10182.581,E2 10182.581} C_VEL
LIN {X 0,Y 556.055,Z 977.53,A -85,B 0,C 180,E1 10187.476,E2 10187.476} C_VEL
LIN {X 0,Y 555.901,Z 977.53,A -85,B 0,C 180,E1 10192.425,E2 10192.425} C_VEL
LIN {X 0,Y 555.748,Z 977.53,A -85,B 0,C 180,E1 10197.606,E2 10197.606} C_VEL
LIN {X 0,Y 555.643,Z 977.53,A -85,B 0,C 180,E1 10203.044,E2 10203.044} C_VEL
LIN {X 0,Y 555.568,Z 977.53,A -85,B 0,C 180,E1 10208.842,E2 10208.842} C_VEL
LIN {X 0,Y 555.547,Z 977.53,A -85,B 0,C 180,E1 10214.825,E2 10214.825} C_VEL
LIN {X 0,Y 555.517,Z 977.53,A -85,B 0,C 180,E1 10219.784,E2 10219.784} C_VEL
LIN {X 0,Y 555.523,Z 977.53,A -85,B 0,C 180,E1 10225.045,E2 10225.045} C_VEL
LIN {X 0,Y 555.781,Z 977.623,A -85,B 0,C 180,E1 10228.573,E2 10228.573} C_VEL
LIN {X 0,Y 574.004,Z 1027.61,A -85,B 0,C 180,E1 10230.451,E2 10230.451} C_VEL
LIN {X 0,Y 574.2,Z 1043.751,A -85,B 0,C 180,E1 10230.951,E2 10230.951} C_VEL
LIN {X 0,Y 571.504,Z 1082.557,A -85,B 0,C 180,E1 10232.443,E2 10232.443} C_VEL
LIN {X 0,Y 568.469,Z 1118.264,A -85,B 0,C 180,E1 10234.43,E2 10234.43} C_VEL
LIN {X 0,Y 565.186,Z 1152.268,A -85,B 0,C 180,E1 10237.01,E2 10237.01} C_VEL
LIN {X 0,Y 562.071,Z 1183.421,A -85,B 0,C 180,E1 10240.209,E2 10240.209} C_VEL
LIN {X 0,Y 559.864,Z 1207.369,A -85,B 0,C 180,E1 10243.498,E2 10243.498} C_VEL
LIN {X 0,Y 558.226,Z 1226.626,A -85,B 0,C 180,E1 10247.05,E2 10247.05} C_VEL
LIN {X 0,Y 557.304,Z 1241.598,A -85,B 0,C 180,E1 10250.995,E2 10250.995} C_VEL
LIN {X 0,Y 556.934,Z 1250.183,A -85,B 0,C 180,E1 10254.525,E2 10254.525} C_VEL
LIN {X 0,Y 556.801,Z 1254.703,A -85,B 0,C 180,E1 10258.43,E2 10258.43} C_VEL
LIN {X 0,Y 556.945,Z 1254.735,A -85,B 0,C 180,E1 10261.548,E2 10261.548} C_VEL
LIN {X 0,Y 557.041,Z 1250.325,A -85,B 0,C 180,E1 10265.451,E2 10265.451} C_VEL
LIN {X 0,Y 557.451,Z 1240.664,A -85,B 0,C 180,E1 10269.374,E2 10269.374} C_VEL
LIN {X 0,Y 558.423,Z 1225.054,A -85,B 0,C 180,E1 10273.322,E2 10273.322} C_VEL
LIN {X 0,Y 560.132,Z 1205.736,A -85,B 0,C 180,E1 10276.772,E2 10276.772} C_VEL
LIN {X 0,Y 562.514,Z 1180.298,A -85,B 0,C 180,E1 10280.139,E2 10280.139} C_VEL
LIN {X 0,Y 565.502,Z 1150.818,A -85,B 0,C 180,E1 10283.057,E2 10283.057} C_VEL
LIN {X 0,Y 568.579,Z 1117.351,A -85,B 0,C 180,E1 10285.541,E2 10285.541} C_VEL
LIN {X 0,Y 571.667,Z 1078.811,A -85,B 0,C 180,E1 10287.611,E2 10287.611} C_VEL
LIN {X 0,Y 574.083,Z 1038.323,A -85,B 0,C 180,E1 10289.067,E2 10289.067} C_VEL
LIN {X 0,Y 573.75,Z 1028.35,A -85,B 0,C 180,E1 10289.378,E2 10289.378} C_VEL
LIN {X 0,Y 562.71,Z 994.164,A -85,B 0,C 180,E1 10290.806,E2 10290.806} C_VEL
LIN {X 0,Y 555.729,Z 977.53,A -85,B 0,C 180,E1 10291.659,E2 10291.659} C_VEL
LIN {X 0,Y 555.518,Z 977.53,A -85,B 0,C 180,E1 10297.731,E2 10297.731} C_VEL
LIN {X 0,Y 555.429,Z 977.53,A -85,B 0,C 180,E1 10302.98,E2 10302.98} C_VEL
LIN {X 0,Y 555.455,Z 977.53,A -85,B 0,C 180,E1 10309.112,E2 10309.112} C_VEL
LIN {X 0,Y 555.606,Z 977.53,A -85,B 0,C 180,E1 10315.069,E2 10315.069} C_VEL
LIN {X 0,Y 555.706,Z 977.53,A -85,B 0,C 180,E1 10316.294,E2 10316.294} C_VEL
LIN {X 0,Y 555.005,Z 981.679,A -85,B 0,C 180,E1 10316.801,E2 10316.801} C_VEL
LIN {X 0,Y 552.217,Z 995.809,A -85,B 0,C 180,E1 10317.581,E2 10317.581} C_VEL
LIN {X 0,Y 552.408,Z 996.917,A -85,B 0,C 180,E1 10317.661,E2 10317.661} C_VEL
LIN {X 0,Y 555.813,Z 1009.55,A -85,B 0,C 180,E1 10318.455,E2 10318.455} C_VEL
LIN {X 0,Y 567.043,Z 1043.191,A -85,B 0,C 180,E1 10319.813,E2 10319.813} C_VEL
LIN {X 0,Y 564.979,Z 1087.775,A -85,B 0,C 180,E1 10320.818,E2 10320.818} C_VEL
LIN {X 0,Y 562.076,Z 1129.718,A -85,B 0,C 180,E1 10322.405,E2 10322.405} C_VEL
LIN {X 0,Y 558.916,Z 1168.645,A -85,B 0,C 180,E1 10324.558,E2 10324.558} C_VEL
LIN {X 0,Y 555.689,Z 1203.964,A -85,B 0,C 180,E1 10327.248,E2 10327.248} C_VEL
LIN {X 0,Y 553.099,Z 1233.03,A -85,B 0,C 180,E1 10330.19,E2 10330.19} C_VEL
LIN {X 0,Y 551.17,Z 1257.473,A -85,B 0,C 180,E1 10333.435,E2 10333.435} C_VEL
LIN {X 0,Y 549.97,Z 1276.952,A -85,B 0,C 180,E1 10336.869,E2 10336.869} C_VEL
LIN {X 0,Y 549.292,Z 1293.01,A -85,B 0,C 180,E1 10340.881,E2 10340.881} C_VEL
LIN {X 0,Y 549.144,Z 1302.197,A -85,B 0,C 180,E1 10344.465,E2 10344.465} C_VEL
LIN {X 0,Y 549.119,Z 1307.06,A -85,B 0,C 180,E1 10348.426,E2 10348.426} C_VEL
LIN {X 0,Y 549.115,Z 1307.133,A -85,B 0,C 180,E1 10351.589,E2 10351.589} C_VEL
LIN {X 0,Y 549.149,Z 1302.493,A -85,B 0,C 180,E1 10355.549,E2 10355.549} C_VEL
LIN {X 0,Y 549.3,Z 1292.32,A -85,B 0,C 180,E1 10359.534,E2 10359.534} C_VEL
LIN {X 0,Y 550.047,Z 1277.963,A -85,B 0,C 180,E1 10363.144,E2 10363.144} C_VEL
LIN {X 0,Y 551.509,Z 1256.42,A -85,B 0,C 180,E1 10366.981,E2 10366.981} C_VEL
LIN {X 0,Y 553.853,Z 1230.095,A -85,B 0,C 180,E1 10370.423,E2 10370.423} C_VEL
LIN {X 0,Y 556.721,Z 1200.313,A -85,B 0,C 180,E1 10373.358,E2 10373.358} C_VEL
LIN {X 0,Y 559.917,Z 1166.455,A -85,B 0,C 180,E1 10375.869,E2 10375.869} C_VEL
LIN {X 0,Y 563.176,Z 1129.198,A -85,B 0,C 180,E1 10377.879,E2 10377.879} C_VEL
LIN {X 0,Y 565.908,Z 1088.796,A -85,B 0,C 180,E1 10379.357,E2 10379.357} C_VEL
LIN {X 0,Y 567.566,Z 1045.844,A -85,B 0,C 180,E1 10380.255,E2 10380.255} C_VEL
LIN {X 0,Y 566.064,Z 1038.833,A -85,B 0,C 180,E1 10380.439,E2 10380.439} C_VEL
LIN {X 0,Y 553.386,Z 999.39,A -85,B 0,C 180,E1 10381.764,E2 10381.764} C_VEL
LIN {X 0,Y 547.79,Z 977.53,A -85,B 0,C 180,E1 10383.598,E2 10383.598} C_VEL
LIN {X 0,Y 547.646,Z 977.53,A -85,B 0,C 180,E1 10389.532,E2 10389.532} C_VEL
LIN {X 0,Y 547.603,Z 977.53,A -85,B 0,C 180,E1 10396.019,E2 10396.019} C_VEL
LIN {X 0,Y 547.592,Z 977.53,A -85,B 0,C 180,E1 10400.798,E2 10400.798} C_VEL
LIN {X 0,Y 547.614,Z 977.53,A -85,B 0,C 180,E1 10406.417,E2 10406.417} C_VEL
LIN {X 0,Y 547.902,Z 977.53,A -85,B 0,C 180,E1 10412.265,E2 10412.265} C_VEL
LIN {X 0,Y 547.986,Z 977.53,A -85,B 0,C 180,E1 10417.24,E2 10417.24} C_VEL
LIN {X 0,Y 548.129,Z 977.53,A -85,B 0,C 180,E1 10422.311,E2 10422.311} C_VEL
LIN {X 0,Y 548.201,Z 977.53,A -85,B 0,C 180,E1 10427.238,E2 10427.238} C_VEL
LIN {X 0,Y 548.341,Z 977.53,A -85,B 0,C 180,E1 10430.419,E2 10430.419} C_VEL
LIN {X 0,Y 560.639,Z 1013.622,A -85,B 0,C 180,E1 10432.157,E2 10432.157} C_VEL
LIN {X 0,Y 558.468,Z 1070.958,A -85,B 0,C 180,E1 10433.594,E2 10433.594} C_VEL
LIN {X 0,Y 557.009,Z 1099.264,A -85,B 0,C 180,E1 10434.94,E2 10434.94} C_VEL
LIN {X 0,Y 555.113,Z 1125.116,A -85,B 0,C 180,E1 10436.882,E2 10436.882} C_VEL
LIN {X 0,Y 553.384,Z 1145.777,A -85,B 0,C 180,E1 10439.193,E2 10439.193} C_VEL
LIN {X 0,Y 551.828,Z 1162.425,A -85,B 0,C 180,E1 10441.978,E2 10441.978} C_VEL
LIN {X 0,Y 550.803,Z 1172.828,A -85,B 0,C 180,E1 10444.745,E2 10444.745} C_VEL
LIN {X 0,Y 550.154,Z 1178.641,A -85,B 0,C 180,E1 10447.926,E2 10447.926} C_VEL
LIN {X 0,Y 550.029,Z 1178.522,A -85,B 0,C 180,E1 10451.129,E2 10451.129} C_VEL
LIN {X 0,Y 550.241,Z 1173.432,A -85,B 0,C 180,E1 10453.953,E2 10453.953} C_VEL
LIN {X 0,Y 550.741,Z 1163.181,A -85,B 0,C 180,E1 10456.801,E2 10456.801} C_VEL
LIN {X 0,Y 551.741,Z 1146.386,A -85,B 0,C 180,E1 10459.669,E2 10459.669} C_VEL
LIN {X 0,Y 553.088,Z 1126.166,A -85,B 0,C 180,E1 10461.985,E2 10461.985} C_VEL
LIN {X 0,Y 554.448,Z 1101.574,A -85,B 0,C 180,E1 10463.921,E2 10463.921} C_VEL
LIN {X 0,Y 555.681,Z 1072.66,A -85,B 0,C 180,E1 10465.39,E2 10465.39} C_VEL
LIN {X 0,Y 556.292,Z 1042.69,A -85,B 0,C 180,E1 10466.233,E2 10466.233} C_VEL
LIN {X 0,Y 556.352,Z 1008.477,A -85,B 0,C 180,E1 10466.855,E2 10466.855} C_VEL
LIN {X 0,Y 547.976,Z 977.53,A -85,B 0,C 180,E1 10467.75,E2 10467.75} C_VEL
LIN {X 0,Y 547.657,Z 977.53,A -85,B 0,C 180,E1 10473.884,E2 10473.884} C_VEL
LIN {X 0,Y 547.658,Z 977.53,A -85,B 0,C 180,E1 10479.53,E2 10479.53} C_VEL
LIN {X 0,Y 547.602,Z 977.53,A -85,B 0,C 180,E1 10486.018,E2 10486.018} C_VEL
LIN {X 0,Y 547.608,Z 977.53,A -85,B 0,C 180,E1 10490.794,E2 10490.794} C_VEL
LIN {X 0,Y 547.62,Z 977.53,A -85,B 0,C 180,E1 10496.391,E2 10496.391} C_VEL
LIN {X 0,Y 547.862,Z 977.53,A -85,B 0,C 180,E1 10502.269,E2 10502.269} C_VEL
LIN {X 0,Y 547.988,Z 977.53,A -85,B 0,C 180,E1 10507.217,E2 10507.217} C_VEL
LIN {X 0,Y 548.134,Z 977.53,A -85,B 0,C 180,E1 10512.289,E2 10512.289} C_VEL
LIN {X 0,Y 548.236,Z 977.53,A -85,B 0,C 180,E1 10517.218,E2 10517.218} C_VEL
LIN {X 0,Y 548.484,Z 977.53,A -85,B 0,C 180,E1 10522.053,E2 10522.053} C_VEL
LIN {X 0,Y 548.641,Z 977.53,A -85,B 0,C 180,E1 10526.826,E2 10526.826} C_VEL
LIN {X 0,Y 548.777,Z 977.53,A -85,B 0,C 180,E1 10531.575,E2 10531.575} C_VEL
LIN {X 0,Y 548.521,Z 977.53,A -85,B 0,C 180,E1 10536.337,E2 10536.337} C_VEL
LIN {X 0,Y 548.297,Z 977.53,A -85,B 0,C 180,E1 10541.147,E2 10541.147} C_VEL
LIN {X 0,Y 548.158,Z 977.53,A -85,B 0,C 180,E1 10546.039,E2 10546.039} C_VEL
LIN {X 0,Y 548.011,Z 977.53,A -85,B 0,C 180,E1 10551.059,E2 10551.059} C_VEL
LIN {X 0,Y 547.846,Z 977.53,A -85,B 0,C 180,E1 10556.258,E2 10556.258} C_VEL
LIN {X 0,Y 547.765,Z 977.53,A -85,B 0,C 180,E1 10561.699,E2 10561.699} C_VEL
LIN {X 0,Y 547.637,Z 977.53,A -85,B 0,C 180,E1 10567.488,E2 10567.488} C_VEL
LIN {X 0,Y 547.603,Z 977.53,A -85,B 0,C 180,E1 10573.76,E2 10573.76} C_VEL
LIN {X 0,Y 547.603,Z 977.53,A -85,B 0,C 180,E1 10578.378,E2 10578.378} C_VEL
LIN {X 0,Y 547.564,Z 977.53,A -85,B 0,C 180,E1 10584.461,E2 10584.461} C_VEL
LIN {X 0,Y 547.812,Z 977.545,A -85,B 0,C 180,E1 10588.153,E2 10588.153} C_VEL
LIN {X 0,Y 566.416,Z 1028.286,A -85,B 0,C 180,E1 10590.105,E2 10590.105} C_VEL
LIN {X 0,Y 567.353,Z 1037.889,A -85,B 0,C 180,E1 10590.43,E2 10590.43} C_VEL
LIN {X 0,Y 564.589,Z 1078.535,A -85,B 0,C 180,E1 10591.926,E2 10591.926} C_VEL
LIN {X 0,Y 561.306,Z 1116.01,A -85,B 0,C 180,E1 10593.972,E2 10593.972} C_VEL
LIN {X 0,Y 558.002,Z 1149.498,A -85,B 0,C 180,E1 10596.485,E2 10596.485} C_VEL
LIN {X 0,Y 554.95,Z 1178.798,A -85,B 0,C 180,E1 10599.409,E2 10599.409} C_VEL
LIN {X 0,Y 552.38,Z 1204.944,A -85,B 0,C 180,E1 10602.881,E2 10602.881} C_VEL
LIN {X 0,Y 550.548,Z 1224.881,A -85,B 0,C 180,E1 10606.461,E2 10606.461} C_VEL
LIN {X 0,Y 549.526,Z 1240.658,A -85,B 0,C 180,E1 10610.467,E2 10610.467} C_VEL
LIN {X 0,Y 549.076,Z 1250.497,A -85,B 0,C 180,E1 10614.447,E2 10614.447} C_VEL
LIN {X 0,Y 548.908,Z 1255.066,A -85,B 0,C 180,E1 10618.407,E2 10618.407} C_VEL
LIN {X 0,Y 549.052,Z 1255.12,A -85,B 0,C 180,E1 10621.57,E2 10621.57} C_VEL
LIN {X 0,Y 549.178,Z 1250.713,A -85,B 0,C 180,E1 10625.53,E2 10625.53} C_VEL
LIN {X 0,Y 549.606,Z 1241.031,A -85,B 0,C 180,E1 10629.509,E2 10629.509} C_VEL
LIN {X 0,Y 550.646,Z 1225.387,A -85,B 0,C 180,E1 10633.514,E2 10633.514} C_VEL
LIN {X 0,Y 552.541,Z 1205.23,A -85,B 0,C 180,E1 10637.133,E2 10637.133} C_VEL
LIN {X 0,Y 555.047,Z 1180.182,A -85,B 0,C 180,E1 10640.463,E2 10640.463} C_VEL
LIN {X 0,Y 558.14,Z 1151.011,A -85,B 0,C 180,E1 10643.379,E2 10643.379} C_VEL
LIN {X 0,Y 561.394,Z 1117.509,A -85,B 0,C 180,E1 10645.892,E2 10645.892} C_VEL
LIN {X 0,Y 564.653,Z 1079.036,A -85,B 0,C 180,E1 10647.979,E2 10647.979} C_VEL
LIN {X 0,Y 567.276,Z 1037.556,A -85,B 0,C 180,E1 10649.482,E2 10649.482} C_VEL
LIN {X 0,Y 566.285,Z 1028.488,A -85,B 0,C 180,E1 10649.814,E2 10649.814} C_VEL
LIN {X 0,Y 556.22,Z 997.03,A -85,B 0,C 180,E1 10651.194,E2 10651.194} C_VEL
LIN {X 0,Y 547.755,Z 977.53,A -85,B 0,C 180,E1 10652.297,E2 10652.297} C_VEL
LIN {X 0,Y 547.609,Z 977.53,A -85,B 0,C 180,E1 10657.48,E2 10657.48} C_VEL
LIN {X 0,Y 547.44,Z 977.53,A -85,B 0,C 180,E1 10663.765,E2 10663.765} C_VEL
LIN {X 0,Y 547.488,Z 977.53,A -85,B 0,C 180,E1 10668.386,E2 10668.386} C_VEL
LIN {X 0,Y 547.69,Z 977.53,A -85,B 0,C 180,E1 10674.489,E2 10674.489} C_VEL
LIN {X 0,Y 547.846,Z 978.236,A -85,B 0,C 180,E1 10676.239,E2 10676.239} C_VEL
LIN {X 0,Y 552.408,Z 996.917,A -85,B 0,C 180,E1 10677.661,E2 10677.661} C_VEL
LIN {X 0,Y 553.5,Z 1008.764,A -85,B 0,C 180,E1 10678.228,E2 10678.228} C_VEL
LIN {X 0,Y 555.024,Z 1030.164,A -85,B 0,C 180,E1 10678.815,E2 10678.815} C_VEL
LIN {X 0,Y 560.237,Z 1047.118,A -85,B 0,C 180,E1 10679.48,E2 10679.48} C_VEL
LIN {X 0,Y 557.824,Z 1090.583,A -85,B 0,C 180,E1 10680.529,E2 10680.529} C_VEL
LIN {X 0,Y 554.726,Z 1132.114,A -85,B 0,C 180,E1 10682.173,E2 10682.173} C_VEL
LIN {X 0,Y 551.414,Z 1169.784,A -85,B 0,C 180,E1 10684.331,E2 10684.331} C_VEL
LIN {X 0,Y 548.106,Z 1204.296,A -85,B 0,C 180,E1 10687.023,E2 10687.023} C_VEL
LIN {X 0,Y 545.302,Z 1234.044,A -85,B 0,C 180,E1 10690.107,E2 10690.107} C_VEL
LIN {X 0,Y 543.298,Z 1258.155,A -85,B 0,C 180,E1 10693.397,E2 10693.397} C_VEL
LIN {X 0,Y 542.009,Z 1278.29,A -85,B 0,C 180,E1 10697.084,E2 10697.084} C_VEL
LIN {X 0,Y 541.427,Z 1292.553,A -85,B 0,C 180,E1 10700.747,E2 10700.747} C_VEL
LIN {X 0,Y 541.268,Z 1301.784,A -85,B 0,C 180,E1 10704.385,E2 10704.385} C_VEL
LIN {X 0,Y 541.223,Z 1306.68,A -85,B 0,C 180,E1 10708.403,E2 10708.403} C_VEL
LIN {X 0,Y 541.219,Z 1306.751,A -85,B 0,C 180,E1 10711.612,E2 10711.612} C_VEL
LIN {X 0,Y 541.275,Z 1302.081,A -85,B 0,C 180,E1 10715.63,E2 10715.63} C_VEL
LIN {X 0,Y 541.429,Z 1291.842,A -85,B 0,C 180,E1 10719.674,E2 10719.674} C_VEL
LIN {X 0,Y 542.261,Z 1276.425,A -85,B 0,C 180,E1 10723.542,E2 10723.542} C_VEL
LIN {X 0,Y 543.923,Z 1254.337,A -85,B 0,C 180,E1 10727.434,E2 10727.434} C_VEL
LIN {X 0,Y 546.243,Z 1229.206,A -85,B 0,C 180,E1 10730.721,E2 10730.721} C_VEL
LIN {X 0,Y 549.231,Z 1199.224,A -85,B 0,C 180,E1 10733.696,E2 10733.696} C_VEL
LIN {X 0,Y 552.544,Z 1165.307,A -85,B 0,C 180,E1 10736.222,E2 10736.222} C_VEL
LIN {X 0,Y 555.935,Z 1127.313,A -85,B 0,C 180,E1 10738.275,E2 10738.275} C_VEL
LIN {X 0,Y 558.874,Z 1085.749,A -85,B 0,C 180,E1 10739.772,E2 10739.772} C_VEL
LIN {X 0,Y 560.13,Z 1043.755,A -85,B 0,C 180,E1 10740.651,E2 10740.651} C_VEL
LIN {X 0,Y 545.718,Z 999.584,A -85,B 0,C 180,E1 10742.171,E2 10742.171} C_VEL
LIN {X 0,Y 539.836,Z 977.53,A -85,B 0,C 180,E1 10744.068,E2 10744.068} C_VEL
LIN {X 0,Y 539.659,Z 977.53,A -85,B 0,C 180,E1 10750.235,E2 10750.235} C_VEL
LIN {X 0,Y 539.65,Z 977.53,A -85,B 0,C 180,E1 10755.438,E2 10755.438} C_VEL
LIN {X 0,Y 539.634,Z 977.53,A -85,B 0,C 180,E1 10761.868,E2 10761.868} C_VEL
LIN {X 0,Y 539.747,Z 977.53,A -85,B 0,C 180,E1 10767.782,E2 10767.782} C_VEL
LIN {X 0,Y 539.998,Z 977.53,A -85,B 0,C 180,E1 10773.905,E2 10773.905} C_VEL
LIN {X 0,Y 540.089,Z 977.53,A -85,B 0,C 180,E1 10778.624,E2 10778.624} C_VEL
LIN {X 0,Y 540.198,Z 977.53,A -85,B 0,C 180,E1 10783.724,E2 10783.724} C_VEL
LIN {X 0,Y 540.385,Z 977.53,A -85,B 0,C 180,E1 10789.904,E2 10789.904} C_VEL
LIN {X 0,Y 553.36,Z 1014.477,A -85,B 0,C 180,E1 10791.775,E2 10791.775} C_VEL
LIN {X 0,Y 551.158,Z 1073.825,A -85,B 0,C 180,E1 10793.352,E2 10793.352} C_VEL
LIN {X 0,Y 549.67,Z 1100.62,A -85,B 0,C 180,E1 10794.674,E2 10794.674} C_VEL
LIN {X 0,Y 547.642,Z 1126.208,A -85,B 0,C 180,E1 10796.641,E2 10796.641} C_VEL
LIN {X 0,Y 545.783,Z 1147.048,A -85,B 0,C 180,E1 10799.017,E2 10799.017} C_VEL
LIN {X 0,Y 544.265,Z 1162.466,A -85,B 0,C 180,E1 10801.607,E2 10801.607} C_VEL
LIN {X 0,Y 543.1,Z 1173.212,A -85,B 0,C 180,E1 10804.411,E2 10804.411} C_VEL
LIN {X 0,Y 542.582,Z 1177.8,A -85,B 0,C 180,E1 10806.424,E2 10806.424} C_VEL
LIN {X 0,Y 542.171,Z 1180.289,A -85,B 0,C 180,E1 10809.664,E2 10809.664} C_VEL
LIN {X 0,Y 542.302,Z 1176.786,A -85,B 0,C 180,E1 10812.927,E2 10812.927} C_VEL
LIN {X 0,Y 542.754,Z 1168.043,A -85,B 0,C 180,E1 10815.919,E2 10815.919} C_VEL
LIN {X 0,Y 543.536,Z 1154.508,A -85,B 0,C 180,E1 10818.673,E2 10818.673} C_VEL
LIN {X 0,Y 544.761,Z 1135.867,A -85,B 0,C 180,E1 10821.208,E2 10821.208} C_VEL
LIN {X 0,Y 546.124,Z 1112.247,A -85,B 0,C 180,E1 10823.399,E2 10823.399} C_VEL
LIN {X 0,Y 547.684,Z 1084.312,A -85,B 0,C 180,E1 10825.114,E2 10825.114} C_VEL
LIN {X 0,Y 548.609,Z 1054.894,A -85,B 0,C 180,E1 10826.191,E2 10826.191} C_VEL
LIN {X 0,Y 548.878,Z 1010.11,A -85,B 0,C 180,E1 10827.072,E2 10827.072} C_VEL
LIN {X 0,Y 540.035,Z 977.53,A -85,B 0,C 180,E1 10828.067,E2 10828.067} C_VEL
LIN {X 0,Y 539.751,Z 977.53,A -85,B 0,C 180,E1 10834.167,E2 10834.167} C_VEL
LIN {X 0,Y 539.677,Z 977.53,A -85,B 0,C 180,E1 10840.233,E2 10840.233} C_VEL
LIN {X 0,Y 539.65,Z 977.53,A -85,B 0,C 180,E1 10845.405,E2 10845.405} C_VEL
LIN {X 0,Y 539.659,Z 977.53,A -85,B 0,C 180,E1 10851.841,E2 10851.841} C_VEL
LIN {X 0,Y 539.738,Z 977.53,A -85,B 0,C 180,E1 10857.755,E2 10857.755} C_VEL
LIN {X 0,Y 539.996,Z 977.53,A -85,B 0,C 180,E1 10863.901,E2 10863.901} C_VEL
LIN {X 0,Y 540.08,Z 977.53,A -85,B 0,C 180,E1 10868.601,E2 10868.601} C_VEL
LIN {X 0,Y 540.213,Z 977.53,A -85,B 0,C 180,E1 10873.703,E2 10873.703} C_VEL
LIN {X 0,Y 540.436,Z 977.53,A -85,B 0,C 180,E1 10878.934,E2 10878.934} C_VEL
LIN {X 0,Y 540.628,Z 977.53,A -85,B 0,C 180,E1 10883.555,E2 10883.555} C_VEL
LIN {X 0,Y 540.74,Z 977.53,A -85,B 0,C 180,E1 10888.387,E2 10888.387} C_VEL
LIN {X 0,Y 540.715,Z 977.53,A -85,B 0,C 180,E1 10893.205,E2 10893.205} C_VEL
LIN {X 0,Y 540.46,Z 977.53,A -85,B 0,C 180,E1 10898.051,E2 10898.051} C_VEL
LIN {X 0,Y 540.325,Z 977.53,A -85,B 0,C 180,E1 10902.957,E2 10902.957} C_VEL
LIN {X 0,Y 540.237,Z 977.53,A -85,B 0,C 180,E1 10907.963,E2 10907.963} C_VEL
LIN {X 0,Y 540.039,Z 977.53,A -85,B 0,C 180,E1 10913.122,E2 10913.122} C_VEL
LIN {X 0,Y 539.859,Z 977.53,A -85,B 0,C 180,E1 10918.491,E2 10918.491} C_VEL
LIN {X 0,Y 539.737,Z 977.53,A -85,B 0,C 180,E1 10924.149,E2 10924.149} C_VEL
LIN {X 0,Y 539.661,Z 977.53,A -85,B 0,C 180,E1 10930.215,E2 10930.215} C_VEL
LIN {X 0,Y 539.621,Z 977.53,A -85,B 0,C 180,E1 10935.403,E2 10935.403} C_VEL
LIN {X 0,Y 539.613,Z 977.53,A -85,B 0,C 180,E1 10939.761,E2 10939.761} C_VEL
LIN {X 0,Y 539.693,Z 977.53,A -85,B 0,C 180,E1 10945.829,E2 10945.829} C_VEL
LIN {X 0,Y 539.889,Z 977.53,A -85,B 0,C 180,E1 10947.713,E2 10947.713} C_VEL
LIN {X 0,Y 558.926,Z 1029.416,A -85,B 0,C 180,E1 10949.77,E2 10949.77} C_VEL
LIN {X 0,Y 560.184,Z 1038.347,A -85,B 0,C 180,E1 10950.098,E2 10950.098} C_VEL
LIN {X 0,Y 557.259,Z 1079.711,A -85,B 0,C 180,E1 10951.651,E2 10951.651} C_VEL
LIN {X 0,Y 553.899,Z 1116.745,A -85,B 0,C 180,E1 10953.706,E2 10953.706} C_VEL
LIN {X 0,Y 550.466,Z 1150.199,A -85,B 0,C 180,E1 10956.251,E2 10956.251} C_VEL
LIN {X 0,Y 547.204,Z 1180.329,A -85,B 0,C 180,E1 10959.316,E2 10959.316} C_VEL
LIN {X 0,Y 544.585,Z 1205.964,A -85,B 0,C 180,E1 10962.795,E2 10962.795} C_VEL
LIN {X 0,Y 542.637,Z 1226.911,A -85,B 0,C 180,E1 10966.671,E2 10966.671} C_VEL
LIN {X 0,Y 541.599,Z 1242.094,A -85,B 0,C 180,E1 10970.732,E2 10970.732} C_VEL
LIN {X 0,Y 541.214,Z 1250.8,A -85,B 0,C 180,E1 10974.366,E2 10974.366} C_VEL
LIN {X 0,Y 541.029,Z 1255.428,A -85,B 0,C 180,E1 10978.384,E2 10978.384} C_VEL
LIN {X 0,Y 541.163,Z 1255.509,A -85,B 0,C 180,E1 10981.593,E2 10981.593} C_VEL
LIN {X 0,Y 541.307,Z 1251.112,A -85,B 0,C 180,E1 10985.61,E2 10985.61} C_VEL
LIN {X 0,Y 541.775,Z 1241.417,A -85,B 0,C 180,E1 10989.648,E2 10989.648} C_VEL
LIN {X 0,Y 542.898,Z 1225.749,A -85,B 0,C 180,E1 10993.71,E2 10993.71} C_VEL
LIN {X 0,Y 544.919,Z 1205.569,A -85,B 0,C 180,E1 10997.379,E2 10997.379} C_VEL
LIN {X 0,Y 547.47,Z 1181.397,A -85,B 0,C 180,E1 11000.649,E2 11000.649} C_VEL
LIN {X 0,Y 550.712,Z 1152.442,A -85,B 0,C 180,E1 11003.606,E2 11003.606} C_VEL
LIN {X 0,Y 554.082,Z 1119.311,A -85,B 0,C 180,E1 11006.15,E2 11006.15} C_VEL
LIN {X 0,Y 557.499,Z 1081.537,A -85,B 0,C 180,E1 11008.262,E2 11008.262} C_VEL
LIN {X 0,Y 560.353,Z 1039.779,A -85,B 0,C 180,E1 11009.832,E2 11009.832} C_VEL
LIN {X 0,Y 559.449,Z 1030.362,A -85,B 0,C 180,E1 11010.189,E2 11010.189} C_VEL
LIN {X 0,Y 550.24,Z 1000.882,A -85,B 0,C 180,E1 11011.547,E2 11011.547} C_VEL
LIN {X 0,Y 539.785,Z 977.53,A -85,B 0,C 180,E1 11012.981,E2 11012.981} C_VEL
LIN {X 0,Y 539.649,Z 977.53,A -85,B 0,C 180,E1 11018.18,E2 11018.18} C_VEL
LIN {X 0,Y 539.475,Z 977.53,A -85,B 0,C 180,E1 11024.58,E2 11024.58} C_VEL
LIN {X 0,Y 539.566,Z 977.53,A -85,B 0,C 180,E1 11029.776,E2 11029.776} C_VEL
LIN {X 0,Y 539.883,Z 977.645,A -85,B 0,C 180,E1 11035.814,E2 11035.814} C_VEL
LIN {X 0,Y 545.684,Z 1000.966,A -85,B 0,C 180,E1 11037.515,E2 11037.515} C_VEL
LIN {X 0,Y 555.024,Z 1030.164,A -85,B 0,C 180,E1 11038.815,E2 11038.815} C_VEL
LIN {X 0,Y 555.79,Z 1043.444,A -85,B 0,C 180,E1 11039.122,E2 11039.122} C_VEL
LIN {X 0,Y 552.632,Z 1065.12,A -85,B 0,C 180,E1 11039.427,E2 11039.427} C_VEL
LIN {X 0,Y 549.613,Z 1108.331,A -85,B 0,C 180,E1 11040.766,E2 11040.766} C_VEL
LIN {X 0,Y 546.024,Z 1148.608,A -85,B 0,C 180,E1 11042.69,E2 11042.69} C_VEL
LIN {X 0,Y 542.581,Z 1184.656,A -85,B 0,C 180,E1 11045.099,E2 11045.099} C_VEL
LIN {X 0,Y 539.332,Z 1216.601,A -85,B 0,C 180,E1 11047.946,E2 11047.946} C_VEL
LIN {X 0,Y 536.764,Z 1243.541,A -85,B 0,C 180,E1 11051.102,E2 11051.102} C_VEL
LIN {X 0,Y 534.888,Z 1266.95,A -85,B 0,C 180,E1 11054.741,E2 11054.741} C_VEL
LIN {X 0,Y 533.892,Z 1284.809,A -85,B 0,C 180,E1 11058.549,E2 11058.549} C_VEL
LIN {X 0,Y 533.429,Z 1297.817,A -85,B 0,C 180,E1 11062.664,E2 11062.664} C_VEL
LIN {X 0,Y 533.298,Z 1304.948,A -85,B 0,C 180,E1 11066.75,E2 11066.75} C_VEL
LIN {X 0,Y 533.343,Z 1306.791,A -85,B 0,C 180,E1 11070.008,E2 11070.008} C_VEL
LIN {X 0,Y 533.342,Z 1304.224,A -85,B 0,C 180,E1 11074.081,E2 11074.081} C_VEL
LIN {X 0,Y 533.477,Z 1296.205,A -85,B 0,C 180,E1 11078.172,E2 11078.172} C_VEL
LIN {X 0,Y 534.061,Z 1281.944,A -85,B 0,C 180,E1 11082.371,E2 11082.371} C_VEL
LIN {X 0,Y 535.354,Z 1262.619,A -85,B 0,C 180,E1 11086.247,E2 11086.247} C_VEL
LIN {X 0,Y 537.533,Z 1238.627,A -85,B 0,C 180,E1 11089.779,E2 11089.779} C_VEL
LIN {X 0,Y 540.516,Z 1209.909,A -85,B 0,C 180,E1 11092.96,E2 11092.96} C_VEL
LIN {X 0,Y 543.992,Z 1177.07,A -85,B 0,C 180,E1 11095.697,E2 11095.697} C_VEL
LIN {X 0,Y 547.463,Z 1141.201,A -85,B 0,C 180,E1 11097.907,E2 11097.907} C_VEL
LIN {X 0,Y 550.627,Z 1102.236,A -85,B 0,C 180,E1 11099.587,E2 11099.587} C_VEL
LIN {X 0,Y 552.985,Z 1060.323,A -85,B 0,C 180,E1 11100.707,E2 11100.707} C_VEL
LIN {X 0,Y 552.556,Z 1044.938,A -85,B 0,C 180,E1 11101.008,E2 11101.008} C_VEL
LIN {X 0,Y 538.083,Z 1000.002,A -85,B 0,C 180,E1 11102.588,E2 11102.588} C_VEL
LIN {X 0,Y 531.878,Z 977.53,A -85,B 0,C 180,E1 11104.625,E2 11104.625} C_VEL
LIN {X 0,Y 531.739,Z 977.53,A -85,B 0,C 180,E1 11110.961,E2 11110.961} C_VEL
LIN {X 0,Y 531.733,Z 977.53,A -85,B 0,C 180,E1 11116.872,E2 11116.872} C_VEL
LIN {X 0,Y 531.659,Z 977.53,A -85,B 0,C 180,E1 11123.256,E2 11123.256} C_VEL
LIN {X 0,Y 531.865,Z 977.53,A -85,B 0,C 180,E1 11129.166,E2 11129.166} C_VEL
LIN {X 0,Y 532.068,Z 977.53,A -85,B 0,C 180,E1 11134.727,E2 11134.727} C_VEL
LIN {X 0,Y 532.213,Z 977.53,A -85,B 0,C 180,E1 11140.037,E2 11140.037} C_VEL
LIN {X 0,Y 532.344,Z 977.53,A -85,B 0,C 180,E1 11145.445,E2 11145.445} C_VEL
LIN {X 0,Y 532.494,Z 977.53,A -85,B 0,C 180,E1 11149.327,E2 11149.327} C_VEL
LIN {X 0,Y 545.887,Z 1014.729,A -85,B 0,C 180,E1 11151.351,E2 11151.351} C_VEL
LIN {X 0,Y 545.923,Z 1029.578,A -85,B 0,C 180,E1 11151.769,E2 11151.769} C_VEL
LIN {X 0,Y 543.881,Z 1076.226,A -85,B 0,C 180,E1 11153.083,E2 11153.083} C_VEL
LIN {X 0,Y 542.145,Z 1104.985,A -85,B 0,C 180,E1 11154.599,E2 11154.599} C_VEL
LIN {X 0,Y 540.033,Z 1129.466,A -85,B 0,C 180,E1 11156.594,E2 11156.594} C_VEL
LIN {X 0,Y 538.01,Z 1149.844,A -85,B 0,C 180,E1 11159.053,E2 11159.053} C_VEL
LIN {X 0,Y 536.486,Z 1164.434,A -85,B 0,C 180,E1 11161.63,E2 11161.63} C_VEL
LIN {X 0,Y 535.28,Z 1174.793,A -85,B 0,C 180,E1 11164.476,E2 11164.476} C_VEL
LIN {X 0,Y 534.618,Z 1180.021,A -85,B 0,C 180,E1 11167.192,E2 11167.192} C_VEL
LIN {X 0,Y 534.343,Z 1181.24,A -85,B 0,C 180,E1 11169.807,E2 11169.807} C_VEL
LIN {X 0,Y 534.488,Z 1177.339,A -85,B 0,C 180,E1 11173.119,E2 11173.119} C_VEL
LIN {X 0,Y 534.995,Z 1168.076,A -85,B 0,C 180,E1 11176.199,E2 11176.199} C_VEL
LIN {X 0,Y 535.914,Z 1153.518,A -85,B 0,C 180,E1 11179.075,E2 11179.075} C_VEL
LIN {X 0,Y 537.3,Z 1133.114,A -85,B 0,C 180,E1 11181.734,E2 11181.734} C_VEL
LIN {X 0,Y 538.68,Z 1109.219,A -85,B 0,C 180,E1 11183.857,E2 11183.857} C_VEL
LIN {X 0,Y 540.236,Z 1080.651,A -85,B 0,C 180,E1 11185.517,E2 11185.517} C_VEL
LIN {X 0,Y 541.065,Z 1050.34,A -85,B 0,C 180,E1 11186.539,E2 11186.539} C_VEL
LIN {X 0,Y 541.178,Z 1010.911,A -85,B 0,C 180,E1 11187.316,E2 11187.316} C_VEL
LIN {X 0,Y 532.086,Z 977.53,A -85,B 0,C 180,E1 11188.336,E2 11188.336} C_VEL
LIN {X 0,Y 531.81,Z 977.53,A -85,B 0,C 180,E1 11194.749,E2 11194.749} C_VEL
LIN {X 0,Y 531.76,Z 977.53,A -85,B 0,C 180,E1 11200.959,E2 11200.959} C_VEL
LIN {X 0,Y 531.738,Z 977.53,A -85,B 0,C 180,E1 11206.839,E2 11206.839} C_VEL
LIN {X 0,Y 531.677,Z 977.53,A -85,B 0,C 180,E1 11213.229,E2 11213.229} C_VEL
LIN {X 0,Y 531.841,Z 977.53,A -85,B 0,C 180,E1 11219.138,E2 11219.138} C_VEL
LIN {X 0,Y 532.057,Z 977.53,A -85,B 0,C 180,E1 11224.702,E2 11224.702} C_VEL
LIN {X 0,Y 532.242,Z 977.53,A -85,B 0,C 180,E1 11230.016,E2 11230.016} C_VEL
LIN {X 0,Y 532.403,Z 977.53,A -85,B 0,C 180,E1 11235.411,E2 11235.411} C_VEL
LIN {X 0,Y 532.66,Z 977.53,A -85,B 0,C 180,E1 11241.815,E2 11241.815} C_VEL
LIN {X 0,Y 532.826,Z 977.53,A -85,B 0,C 180,E1 11246.732,E2 11246.732} C_VEL
LIN {X 0,Y 532.968,Z 977.53,A -85,B 0,C 180,E1 11251.622,E2 11251.622} C_VEL
LIN {X 0,Y 532.682,Z 977.53,A -85,B 0,C 180,E1 11256.526,E2 11256.526} C_VEL
LIN {X 0,Y 532.475,Z 977.53,A -85,B 0,C 180,E1 11261.482,E2 11261.482} C_VEL
LIN {X 0,Y 532.34,Z 977.53,A -85,B 0,C 180,E1 11266.529,E2 11266.529} C_VEL
LIN {X 0,Y 532.165,Z 977.53,A -85,B 0,C 180,E1 11271.717,E2 11271.717} C_VEL
LIN {X 0,Y 531.925,Z 977.53,A -85,B 0,C 180,E1 11277.972,E2 11277.972} C_VEL
LIN {X 0,Y 531.853,Z 977.53,A -85,B 0,C 180,E1 11284.277,E2 11284.277} C_VEL
LIN {X 0,Y 531.701,Z 977.53,A -85,B 0,C 180,E1 11289.685,E2 11289.685} C_VEL
LIN {X 0,Y 531.718,Z 977.53,A -85,B 0,C 180,E1 11295.423,E2 11295.423} C_VEL
LIN {X 0,Y 531.675,Z 977.53,A -85,B 0,C 180,E1 11301.162,E2 11301.162} C_VEL
LIN {X 0,Y 531.935,Z 977.53,A -85,B 0,C 180,E1 11307.268,E2 11307.268} C_VEL
LIN {X 0,Y 551.164,Z 1029.618,A -85,B 0,C 180,E1 11309.391,E2 11309.391} C_VEL
LIN {X 0,Y 553.022,Z 1039.066,A -85,B 0,C 180,E1 11309.769,E2 11309.769} C_VEL
LIN {X 0,Y 549.994,Z 1080.167,A -85,B 0,C 180,E1 11311.335,E2 11311.335} C_VEL
LIN {X 0,Y 546.486,Z 1117.573,A -85,B 0,C 180,E1 11313.442,E2 11313.442} C_VEL
LIN {X 0,Y 542.945,Z 1150.81,A -85,B 0,C 180,E1 11316.011,E2 11316.011} C_VEL
LIN {X 0,Y 539.648,Z 1180.045,A -85,B 0,C 180,E1 11319.013,E2 11319.013} C_VEL
LIN {X 0,Y 536.916,Z 1205.896,A -85,B 0,C 180,E1 11322.541,E2 11322.541} C_VEL
LIN {X 0,Y 534.835,Z 1227.015,A -85,B 0,C 180,E1 11326.473,E2 11326.473} C_VEL
LIN {X 0,Y 533.77,Z 1242.321,A -85,B 0,C 180,E1 11330.595,E2 11330.595} C_VEL
LIN {X 0,Y 533.319,Z 1251.445,A -85,B 0,C 180,E1 11334.47,E2 11334.47} C_VEL
LIN {X 0,Y 533.137,Z 1255.788,A -85,B 0,C 180,E1 11338.36,E2 11338.36} C_VEL
LIN {X 0,Y 533.27,Z 1255.905,A -85,B 0,C 180,E1 11341.616,E2 11341.616} C_VEL
LIN {X 0,Y 533.447,Z 1250.474,A -85,B 0,C 180,E1 11346.256,E2 11346.256} C_VEL
LIN {X 0,Y 534.028,Z 1240.507,A -85,B 0,C 180,E1 11350.202,E2 11350.202} C_VEL
LIN {X 0,Y 535.131,Z 1226.155,A -85,B 0,C 180,E1 11353.913,E2 11353.913} C_VEL
LIN {X 0,Y 537.299,Z 1205.951,A -85,B 0,C 180,E1 11357.634,E2 11357.634} C_VEL
LIN {X 0,Y 540.003,Z 1181.765,A -85,B 0,C 180,E1 11360.948,E2 11360.948} C_VEL
LIN {X 0,Y 543.547,Z 1151.664,A -85,B 0,C 180,E1 11364.045,E2 11364.045} C_VEL
LIN {X 0,Y 547.163,Z 1118.212,A -85,B 0,C 180,E1 11366.617,E2 11366.617} C_VEL
LIN {X 0,Y 550.783,Z 1079.632,A -85,B 0,C 180,E1 11368.762,E2 11368.762} C_VEL
LIN {X 0,Y 553.68,Z 1039.049,A -85,B 0,C 180,E1 11370.286,E2 11370.286} C_VEL
LIN {X 0,Y 546.942,Z 1011.698,A -85,B 0,C 180,E1 11371.548,E2 11371.548} C_VEL
LIN {X 0,Y 535.835,Z 986.788,A -85,B 0,C 180,E1 11373.051,E2 11373.051} C_VEL
LIN {X 0,Y 531.846,Z 977.53,A -85,B 0,C 180,E1 11373.678,E2 11373.678} C_VEL
LIN {X 0,Y 531.623,Z 977.53,A -85,B 0,C 180,E1 11379.697,E2 11379.697} C_VEL
LIN {X 0,Y 531.573,Z 977.53,A -85,B 0,C 180,E1 11385.426,E2 11385.426} C_VEL
LIN {X 0,Y 531.681,Z 977.53,A -85,B 0,C 180,E1 11391.182,E2 11391.182} C_VEL
LIN {X 0,Y 531.934,Z 977.783,A -85,B 0,C 180,E1 11395.433,E2 11395.433} C_VEL
LIN {X 0,Y 536.207,Z 993.661,A -85,B 0,C 180,E1 11396.539,E2 11396.539} C_VEL
LIN {X 0,Y 553.328,Z 1047.515,A -85,B 0,C 180,E1 11399.05,E2 11399.05} C_VEL
LIN {X 0,Y 552.632,Z 1065.12,A -85,B 0,C 180,E1 11399.427,E2 11399.427} C_VEL
LIN {X 0,Y 548.069,Z 1081.953,A -85,B 0,C 180,E1 11399.65,E2 11399.65} C_VEL
LIN {X 0,Y 543.431,Z 1098.474,A -85,B 0,C 180,E1 11399.994,E2 11399.994} C_VEL
LIN {X 0,Y 539.957,Z 1137.621,A -85,B 0,C 180,E1 11401.726,E2 11401.726} C_VEL
LIN {X 0,Y 536.385,Z 1173.281,A -85,B 0,C 180,E1 11403.928,E2 11403.928} C_VEL
LIN {X 0,Y 532.665,Z 1208.035,A -85,B 0,C 180,E1 11406.819,E2 11406.819} C_VEL
LIN {X 0,Y 529.527,Z 1238.412,A -85,B 0,C 180,E1 11410.203,E2 11410.203} C_VEL
LIN {X 0,Y 527.374,Z 1262.126,A -85,B 0,C 180,E1 11413.73,E2 11413.73} C_VEL
LIN {X 0,Y 526.134,Z 1281.028,A -85,B 0,C 180,E1 11417.535,E2 11417.535} C_VEL
LIN {X 0,Y 525.586,Z 1295.315,A -85,B 0,C 180,E1 11421.72,E2 11421.72} C_VEL
LIN {X 0,Y 525.428,Z 1303.607,A -85,B 0,C 180,E1 11425.873,E2 11425.873} C_VEL
LIN {X 0,Y 525.471,Z 1306.407,A -85,B 0,C 180,E1 11430.008,E2 11430.008} C_VEL
LIN {X 0,Y 525.445,Z 1303.817,A -85,B 0,C 180,E1 11434.142,E2 11434.142} C_VEL
LIN {X 0,Y 525.582,Z 1295.741,A -85,B 0,C 180,E1 11438.296,E2 11438.296} C_VEL
LIN {X 0,Y 526.213,Z 1281.715,A -85,B 0,C 180,E1 11442.479,E2 11442.479} C_VEL
LIN {X 0,Y 527.544,Z 1261.891,A -85,B 0,C 180,E1 11446.495,E2 11446.495} C_VEL
LIN {X 0,Y 529.883,Z 1237.717,A -85,B 0,C 180,E1 11450.077,E2 11450.077} C_VEL
LIN {X 0,Y 533.068,Z 1208.5,A -85,B 0,C 180,E1 11453.33,E2 11453.33} C_VEL
LIN {X 0,Y 536.647,Z 1175.632,A -85,B 0,C 180,E1 11456.075,E2 11456.075} C_VEL
LIN {X 0,Y 540.237,Z 1139.817,A -85,B 0,C 180,E1 11458.285,E2 11458.285} C_VEL
LIN {X 0,Y 543.57,Z 1099.705,A -85,B 0,C 180,E1 11460.01,E2 11460.01} C_VEL
LIN {X 0,Y 545.92,Z 1058.499,A -85,B 0,C 180,E1 11461.09,E2 11461.09} C_VEL
LIN {X 0,Y 545.276,Z 1046.708,A -85,B 0,C 180,E1 11461.345,E2 11461.345} C_VEL
LIN {X 0,Y 530.511,Z 1000.729,A -85,B 0,C 180,E1 11463.006,E2 11463.006} C_VEL
LIN {X 0,Y 523.893,Z 977.53,A -85,B 0,C 180,E1 11465.179,E2 11465.179} C_VEL
LIN {X 0,Y 523.826,Z 977.53,A -85,B 0,C 180,E1 11471.253,E2 11471.253} C_VEL
LIN {X 0,Y 523.825,Z 977.53,A -85,B 0,C 180,E1 11476.328,E2 11476.328} C_VEL
LIN {X 0,Y 523.76,Z 977.53,A -85,B 0,C 180,E1 11482.608,E2 11482.608} C_VEL
LIN {X 0,Y 523.935,Z 977.53,A -85,B 0,C 180,E1 11488.647,E2 11488.647} C_VEL
LIN {X 0,Y 524.109,Z 977.53,A -85,B 0,C 180,E1 11494.316,E2 11494.316} C_VEL
LIN {X 0,Y 524.311,Z 977.53,A -85,B 0,C 180,E1 11499.723,E2 11499.723} C_VEL
LIN {X 0,Y 524.405,Z 977.53,A -85,B 0,C 180,E1 11504.941,E2 11504.941} C_VEL
LIN {X 0,Y 524.63,Z 978.298,A -85,B 0,C 180,E1 11508.747,E2 11508.747} C_VEL
LIN {X 0,Y 538.048,Z 1013.558,A -85,B 0,C 180,E1 11510.831,E2 11510.831} C_VEL
LIN {X 0,Y 539.475,Z 1022.107,A -85,B 0,C 180,E1 11511.175,E2 11511.175} C_VEL
LIN {X 0,Y 536.77,Z 1076.371,A -85,B 0,C 180,E1 11512.714,E2 11512.714} C_VEL
LIN {X 0,Y 535.045,Z 1103.434,A -85,B 0,C 180,E1 11514.12,E2 11514.12} C_VEL
LIN {X 0,Y 532.656,Z 1129.685,A -85,B 0,C 180,E1 11516.24,E2 11516.24} C_VEL
LIN {X 0,Y 530.547,Z 1150.098,A -85,B 0,C 180,E1 11518.707,E2 11518.707} C_VEL
LIN {X 0,Y 528.734,Z 1166.403,A -85,B 0,C 180,E1 11521.654,E2 11521.654} C_VEL
LIN {X 0,Y 527.35,Z 1177.326,A -85,B 0,C 180,E1 11524.956,E2 11524.956} C_VEL
LIN {X 0,Y 526.63,Z 1182.03,A -85,B 0,C 180,E1 11528.282,E2 11528.282} C_VEL
LIN {X 0,Y 526.565,Z 1180.752,A -85,B 0,C 180,E1 11531.631,E2 11531.631} C_VEL
LIN {X 0,Y 526.935,Z 1173.4,A -85,B 0,C 180,E1 11535.01,E2 11535.01} C_VEL
LIN {X 0,Y 527.744,Z 1159.958,A -85,B 0,C 180,E1 11538.205,E2 11538.205} C_VEL
LIN {X 0,Y 528.987,Z 1141.294,A -85,B 0,C 180,E1 11541.03,E2 11541.03} C_VEL
LIN {X 0,Y 530.462,Z 1118.541,A -85,B 0,C 180,E1 11543.359,E2 11543.359} C_VEL
LIN {X 0,Y 532.101,Z 1091.702,A -85,B 0,C 180,E1 11545.206,E2 11545.206} C_VEL
LIN {X 0,Y 533.251,Z 1061.685,A -85,B 0,C 180,E1 11546.477,E2 11546.477} C_VEL
LIN {X 0,Y 533.809,Z 1012.927,A -85,B 0,C 180,E1 11547.528,E2 11547.528} C_VEL
LIN {X 0,Y 524.119,Z 977.53,A -85,B 0,C 180,E1 11548.678,E2 11548.678} C_VEL
LIN {X 0,Y 523.936,Z 977.53,A -85,B 0,C 180,E1 11553.342,E2 11553.342} C_VEL
LIN {X 0,Y 523.819,Z 977.53,A -85,B 0,C 180,E1 11559.534,E2 11559.534} C_VEL
LIN {X 0,Y 523.808,Z 977.53,A -85,B 0,C 180,E1 11566.021,E2 11566.021} C_VEL
LIN {X 0,Y 523.741,Z 977.53,A -85,B 0,C 180,E1 11571.377,E2 11571.377} C_VEL
LIN {X 0,Y 523.904,Z 977.53,A -85,B 0,C 180,E1 11577.02,E2 11577.02} C_VEL
LIN {X 0,Y 524.071,Z 977.53,A -85,B 0,C 180,E1 11582.436,E2 11582.436} C_VEL
LIN {X 0,Y 524.23,Z 977.53,A -85,B 0,C 180,E1 11587.921,E2 11587.921} C_VEL
LIN {X 0,Y 524.385,Z 977.53,A -85,B 0,C 180,E1 11593.196,E2 11593.196} C_VEL
LIN {X 0,Y 524.571,Z 977.53,A -85,B 0,C 180,E1 11599.175,E2 11599.175} C_VEL
LIN {X 0,Y 524.878,Z 977.53,A -85,B 0,C 180,E1 11605.024,E2 11605.024} C_VEL
LIN {X 0,Y 525.038,Z 977.53,A -85,B 0,C 180,E1 11609.992,E2 11609.992} C_VEL
LIN {X 0,Y 524.898,Z 977.53,A -85,B 0,C 180,E1 11614.96,E2 11614.96} C_VEL
LIN {X 0,Y 524.558,Z 977.53,A -85,B 0,C 180,E1 11620.818,E2 11620.818} C_VEL
LIN {X 0,Y 524.403,Z 977.53,A -85,B 0,C 180,E1 11626.787,E2 11626.787} C_VEL
LIN {X 0,Y 524.192,Z 977.53,A -85,B 0,C 180,E1 11632.315,E2 11632.315} C_VEL
LIN {X 0,Y 524.05,Z 977.53,A -85,B 0,C 180,E1 11637.548,E2 11637.548} C_VEL
LIN {X 0,Y 523.92,Z 977.53,A -85,B 0,C 180,E1 11643.324,E2 11643.324} C_VEL
LIN {X 0,Y 523.797,Z 977.53,A -85,B 0,C 180,E1 11649.516,E2 11649.516} C_VEL
LIN {X 0,Y 523.791,Z 977.53,A -85,B 0,C 180,E1 11656.019,E2 11656.019} C_VEL
LIN {X 0,Y 523.752,Z 977.53,A -85,B 0,C 180,E1 11661.352,E2 11661.352} C_VEL
LIN {X 0,Y 523.969,Z 977.53,A -85,B 0,C 180,E1 11666.835,E2 11666.835} C_VEL
LIN {X 0,Y 543.443,Z 1030.002,A -85,B 0,C 180,E1 11669.01,E2 11669.01} C_VEL
LIN {X 0,Y 545.877,Z 1039.329,A -85,B 0,C 180,E1 11669.422,E2 11669.422} C_VEL
LIN {X 0,Y 542.814,Z 1079.779,A -85,B 0,C 180,E1 11670.977,E2 11670.977} C_VEL
LIN {X 0,Y 539.202,Z 1116.93,A -85,B 0,C 180,E1 11673.077,E2 11673.077} C_VEL
LIN {X 0,Y 535.567,Z 1150.236,A -85,B 0,C 180,E1 11675.659,E2 11675.659} C_VEL
LIN {X 0,Y 532.121,Z 1179.728,A -85,B 0,C 180,E1 11678.701,E2 11678.701} C_VEL
LIN {X 0,Y 529.217,Z 1205.773,A -85,B 0,C 180,E1 11682.279,E2 11682.279} C_VEL
LIN {X 0,Y 527.063,Z 1227.095,A -85,B 0,C 180,E1 11686.269,E2 11686.269} C_VEL
LIN {X 0,Y 525.929,Z 1242.541,A -85,B 0,C 180,E1 11690.453,E2 11690.453} C_VEL
LIN {X 0,Y 525.446,Z 1251.095,A -85,B 0,C 180,E1 11694.045,E2 11694.045} C_VEL
LIN {X 0,Y 525.258,Z 1256.147,A -85,B 0,C 180,E1 11698.335,E2 11698.335} C_VEL
LIN {X 0,Y 525.383,Z 1256.306,A -85,B 0,C 180,E1 11701.641,E2 11701.641} C_VEL
LIN {X 0,Y 525.583,Z 1251.443,A -85,B 0,C 180,E1 11706.053,E2 11706.053} C_VEL
LIN {X 0,Y 526.117,Z 1242.268,A -85,B 0,C 180,E1 11709.938,E2 11709.938} C_VEL
LIN {X 0,Y 527.41,Z 1226.589,A -85,B 0,C 180,E1 11714.121,E2 11714.121} C_VEL
LIN {X 0,Y 529.681,Z 1206.389,A -85,B 0,C 180,E1 11717.896,E2 11717.896} C_VEL
LIN {X 0,Y 532.564,Z 1182.204,A -85,B 0,C 180,E1 11721.255,E2 11721.255} C_VEL
LIN {X 0,Y 536.277,Z 1152.136,A -85,B 0,C 180,E1 11724.392,E2 11724.392} C_VEL
LIN {X 0,Y 540.262,Z 1117.54,A -85,B 0,C 180,E1 11727.077,E2 11727.077} C_VEL
LIN {X 0,Y 544.056,Z 1079.25,A -85,B 0,C 180,E1 11729.21,E2 11729.21} C_VEL
LIN {X 0,Y 546.791,Z 1037.816,A -85,B 0,C 180,E1 11730.802,E2 11730.802} C_VEL
LIN {X 0,Y 538.522,Z 1008.818,A -85,B 0,C 180,E1 11732.285,E2 11732.285} C_VEL
LIN {X 0,Y 526.24,Z 983.102,A -85,B 0,C 180,E1 11734.085,E2 11734.085} C_VEL
LIN {X 0,Y 523.899,Z 977.53,A -85,B 0,C 180,E1 11734.542,E2 11734.542} C_VEL
LIN {X 0,Y 523.723,Z 977.53,A -85,B 0,C 180,E1 11739.512,E2 11739.512} C_VEL
LIN {X 0,Y 523.65,Z 977.53,A -85,B 0,C 180,E1 11746.025,E2 11746.025} C_VEL
LIN {X 0,Y 523.769,Z 977.53,A -85,B 0,C 180,E1 11751.335,E2 11751.335} C_VEL
LIN {X 0,Y 523.933,Z 977.626,A -85,B 0,C 180,E1 11754.843,E2 11754.843} C_VEL
LIN {X 0,Y 535.546,Z 1013.218,A -85,B 0,C 180,E1 11756.966,E2 11756.966} C_VEL
LIN {X 0,Y 546.711,Z 1051.169,A -85,B 0,C 180,E1 11758.685,E2 11758.685} C_VEL
LIN {X 0,Y 543.65,Z 1095.836,A -85,B 0,C 180,E1 11759.896,E2 11759.896} C_VEL
LIN {X 0,Y 543.431,Z 1098.474,A -85,B 0,C 180,E1 11759.994,E2 11759.994} C_VEL
LIN {X 0,Y 538.607,Z 1114.831,A -85,B 0,C 180,E1 11760.437,E2 11760.437} C_VEL
LIN {X 0,Y 533.57,Z 1130.822,A -85,B 0,C 180,E1 11760.972,E2 11760.972} C_VEL
LIN {X 0,Y 529.479,Z 1169.853,A -85,B 0,C 180,E1 11763.333,E2 11763.333} C_VEL
LIN {X 0,Y 525.483,Z 1204.67,A -85,B 0,C 180,E1 11766.199,E2 11766.199} C_VEL
LIN {X 0,Y 522.304,Z 1234.013,A -85,B 0,C 180,E1 11769.413,E2 11769.413} C_VEL
LIN {X 0,Y 519.856,Z 1259.129,A -85,B 0,C 180,E1 11773.062,E2 11773.062} C_VEL
LIN {X 0,Y 518.417,Z 1278.727,A -85,B 0,C 180,E1 11776.916,E2 11776.916} C_VEL
LIN {X 0,Y 517.765,Z 1292.503,A -85,B 0,C 180,E1 11780.745,E2 11780.745} C_VEL
LIN {X 0,Y 517.576,Z 1301.97,A -85,B 0,C 180,E1 11784.969,E2 11784.969} C_VEL
LIN {X 0,Y 517.536,Z 1305.546,A -85,B 0,C 180,E1 11788.33,E2 11788.33} C_VEL
LIN {X 0,Y 517.534,Z 1305.576,A -85,B 0,C 180,E1 11791.686,E2 11791.686} C_VEL
LIN {X 0,Y 517.605,Z 1301.089,A -85,B 0,C 180,E1 11795.728,E2 11795.728} C_VEL
LIN {X 0,Y 517.76,Z 1291.664,A -85,B 0,C 180,E1 11799.696,E2 11799.696} C_VEL
LIN {X 0,Y 518.74,Z 1275.568,A -85,B 0,C 180,E1 11803.953,E2 11803.953} C_VEL
LIN {X 0,Y 520.493,Z 1254.789,A -85,B 0,C 180,E1 11807.807,E2 11807.807} C_VEL
LIN {X 0,Y 523.275,Z 1228.114,A -85,B 0,C 180,E1 11811.452,E2 11811.452} C_VEL
LIN {X 0,Y 526.61,Z 1197.722,A -85,B 0,C 180,E1 11814.572,E2 11814.572} C_VEL
LIN {X 0,Y 530.402,Z 1163.367,A -85,B 0,C 180,E1 11817.208,E2 11817.208} C_VEL
LIN {X 0,Y 534.223,Z 1124.497,A -85,B 0,C 180,E1 11819.36,E2 11819.36} C_VEL
LIN {X 0,Y 537.413,Z 1083.395,A -85,B 0,C 180,E1 11820.86,E2 11820.86} C_VEL
LIN {X 0,Y 538.304,Z 1049.076,A -85,B 0,C 180,E1 11821.658,E2 11821.658} C_VEL
LIN {X 0,Y 523.318,Z 1002.768,A -85,B 0,C 180,E1 11823.329,E2 11823.329} C_VEL
LIN {X 0,Y 515.93,Z 977.53,A -85,B 0,C 180,E1 11825.818,E2 11825.818} C_VEL
LIN {X 0,Y 515.853,Z 977.53,A -85,B 0,C 180,E1 11832.511,E2 11832.511} C_VEL
LIN {X 0,Y 515.831,Z 977.53,A -85,B 0,C 180,E1 11837.519,E2 11837.519} C_VEL
LIN {X 0,Y 515.844,Z 977.53,A -85,B 0,C 180,E1 11844.041,E2 11844.041} C_VEL
LIN {X 0,Y 516.054,Z 977.53,A -85,B 0,C 180,E1 11850.073,E2 11850.073} C_VEL
LIN {X 0,Y 516.232,Z 977.53,A -85,B 0,C 180,E1 11855.753,E2 11855.753} C_VEL
LIN {X 0,Y 516.384,Z 977.53,A -85,B 0,C 180,E1 11861.184,E2 11861.184} C_VEL
LIN {X 0,Y 516.546,Z 977.53,A -85,B 0,C 180,E1 11867.304,E2 11867.304} C_VEL
LIN {X 0,Y 516.607,Z 977.781,A -85,B 0,C 180,E1 11868.058,E2 11868.058} C_VEL
LIN {X 0,Y 530.792,Z 1014.358,A -85,B 0,C 180,E1 11870.38,E2 11870.38} C_VEL
LIN {X 0,Y 532.565,Z 1023.569,A -85,B 0,C 180,E1 11870.784,E2 11870.784} C_VEL
LIN {X 0,Y 529.645,Z 1077.151,A -85,B 0,C 180,E1 11872.358,E2 11872.358} C_VEL
LIN {X 0,Y 527.771,Z 1104.99,A -85,B 0,C 180,E1 11873.832,E2 11873.832} C_VEL
LIN {X 0,Y 525.239,Z 1130.954,A -85,B 0,C 180,E1 11875.98,E2 11875.98} C_VEL
LIN {X 0,Y 522.965,Z 1151.495,A -85,B 0,C 180,E1 11878.52,E2 11878.52} C_VEL
LIN {X 0,Y 521.182,Z 1166.539,A -85,B 0,C 180,E1 11881.261,E2 11881.261} C_VEL
LIN {X 0,Y 519.791,Z 1176.806,A -85,B 0,C 180,E1 11884.191,E2 11884.191} C_VEL
LIN {X 0,Y 519.028,Z 1181.917,A -85,B 0,C 180,E1 11886.909,E2 11886.909} C_VEL
LIN {X 0,Y 518.661,Z 1183.013,A -85,B 0,C 180,E1 11890.106,E2 11890.106} C_VEL
LIN {X 0,Y 518.869,Z 1178.397,A -85,B 0,C 180,E1 11893.521,E2 11893.521} C_VEL
LIN {X 0,Y 519.394,Z 1168.755,A -85,B 0,C 180,E1 11896.587,E2 11896.587} C_VEL
LIN {X 0,Y 520.446,Z 1153.383,A -85,B 0,C 180,E1 11899.572,E2 11899.572} C_VEL
LIN {X 0,Y 521.93,Z 1133.294,A -85,B 0,C 180,E1 11902.184,E2 11902.184} C_VEL
LIN {X 0,Y 523.55,Z 1108.033,A -85,B 0,C 180,E1 11904.412,E2 11904.412} C_VEL
LIN {X 0,Y 525.069,Z 1079.797,A -85,B 0,C 180,E1 11906.041,E2 11906.041} C_VEL
LIN {X 0,Y 525.976,Z 1048.981,A -85,B 0,C 180,E1 11907.057,E2 11907.057} C_VEL
LIN {X 0,Y 526.223,Z 1014.117,A -85,B 0,C 180,E1 11907.772,E2 11907.772} C_VEL
LIN {X 0,Y 516.213,Z 977.53,A -85,B 0,C 180,E1 11908.937,E2 11908.937} C_VEL
LIN {X 0,Y 515.888,Z 977.53,A -85,B 0,C 180,E1 11914.659,E2 11914.659} C_VEL
LIN {X 0,Y 515.905,Z 977.53,A -85,B 0,C 180,E1 11920.263,E2 11920.263} C_VEL
LIN {X 0,Y 515.834,Z 977.53,A -85,B 0,C 180,E1 11925.159,E2 11925.159} C_VEL
LIN {X 0,Y 515.836,Z 977.53,A -85,B 0,C 180,E1 11929.806,E2 11929.806} C_VEL
LIN {X 0,Y 515.885,Z 977.53,A -85,B 0,C 180,E1 11936.068,E2 11936.068} C_VEL
LIN {X 0,Y 516.089,Z 977.53,A -85,B 0,C 180,E1 11941.972,E2 11941.972} C_VEL
LIN {X 0,Y 516.308,Z 977.53,A -85,B 0,C 180,E1 11947.563,E2 11947.563} C_VEL
LIN {X 0,Y 516.472,Z 977.53,A -85,B 0,C 180,E1 11952.931,E2 11952.931} C_VEL
LIN {X 0,Y 516.626,Z 977.53,A -85,B 0,C 180,E1 11958.144,E2 11958.144} C_VEL
LIN {X 0,Y 516.899,Z 977.53,A -85,B 0,C 180,E1 11963.258,E2 11963.258} C_VEL
LIN {X 0,Y 517.031,Z 977.53,A -85,B 0,C 180,E1 11968.313,E2 11968.313} C_VEL
LIN {X 0,Y 517.013,Z 977.53,A -85,B 0,C 180,E1 11973.353,E2 11973.353} C_VEL
LIN {X 0,Y 516.732,Z 977.53,A -85,B 0,C 180,E1 11978.423,E2 11978.423} C_VEL
LIN {X 0,Y 516.499,Z 977.53,A -85,B 0,C 180,E1 11984.483,E2 11984.483} C_VEL
LIN {X 0,Y 516.371,Z 977.53,A -85,B 0,C 180,E1 11990.609,E2 11990.609} C_VEL
LIN {X 0,Y 516.132,Z 977.53,A -85,B 0,C 180,E1 11996.119,E2 11996.119} C_VEL
LIN {X 0,Y 516.015,Z 977.53,A -85,B 0,C 180,E1 12001.899,E2 12001.899} C_VEL
LIN {X 0,Y 515.888,Z 977.53,A -85,B 0,C 180,E1 12008.074,E2 12008.074} C_VEL
LIN {X 0,Y 515.845,Z 977.53,A -85,B 0,C 180,E1 12012.736,E2 12012.736} C_VEL
LIN {X 0,Y 515.823,Z 977.53,A -85,B 0,C 180,E1 12017.486,E2 12017.486} C_VEL
LIN {X 0,Y 515.851,Z 977.53,A -85,B 0,C 180,E1 12024.012,E2 12024.012} C_VEL
LIN {X 0,Y 515.981,Z 977.53,A -85,B 0,C 180,E1 12026.371,E2 12026.371} C_VEL
LIN {X 0,Y 535.83,Z 1030.73,A -85,B 0,C 180,E1 12028.643,E2 12028.643} C_VEL
LIN {X 0,Y 538.545,Z 1041.854,A -85,B 0,C 180,E1 12029.14,E2 12029.14} C_VEL
LIN {X 0,Y 535.446,Z 1081.468,A -85,B 0,C 180,E1 12030.713,E2 12030.713} C_VEL
LIN {X 0,Y 531.696,Z 1118.59,A -85,B 0,C 180,E1 12032.862,E2 12032.862} C_VEL
LIN {X 0,Y 527.914,Z 1151.919,A -85,B 0,C 180,E1 12035.509,E2 12035.509} C_VEL
LIN {X 0,Y 524.366,Z 1181.141,A -85,B 0,C 180,E1 12038.593,E2 12038.593} C_VEL
LIN {X 0,Y 521.416,Z 1206.993,A -85,B 0,C 180,E1 12042.223,E2 12042.223} C_VEL
LIN {X 0,Y 519.307,Z 1227.136,A -85,B 0,C 180,E1 12046.06,E2 12046.06} C_VEL
LIN {X 0,Y 518.084,Z 1242.736,A -85,B 0,C 180,E1 12050.307,E2 12050.307} C_VEL
LIN {X 0,Y 517.525,Z 1252.304,A -85,B 0,C 180,E1 12054.472,E2 12054.472} C_VEL
LIN {X 0,Y 517.365,Z 1256.504,A -85,B 0,C 180,E1 12058.31,E2 12058.31} C_VEL
LIN {X 0,Y 517.491,Z 1256.712,A -85,B 0,C 180,E1 12061.666,E2 12061.666} C_VEL
LIN {X 0,Y 517.674,Z 1252.687,A -85,B 0,C 180,E1 12065.696,E2 12065.696} C_VEL
LIN {X 0,Y 518.294,Z 1242.725,A -85,B 0,C 180,E1 12070.089,E2 12070.089} C_VEL
